SPLINE
SPL {X  -153.420, Y  +337.122, Z    +0.000, E1  +333.501, E3 -340615.542}
SPL {X  -157.288, Y  +353.220, Z    +0.000, E1  +341.134, E3 -340627.588}
SPL {X  -159.049, Y  +365.172, Z    +0.000, E1  +347.392, E3 -340633.141}
SPL {X  -159.749, Y  +373.719, Z    +0.000, E1  +352.250, E3 -340635.761}
SPL {X  -159.988, Y  +381.741, Z    +0.000, E1  +357.172, E3 -340637.236}
SPL {X  -159.990, Y  +387.352, Z    +0.000, E1  +361.387, E3 -340637.938}
SPL {X  -159.990, Y  +391.188, Z    +0.000, E1  +365.082, E3 -340638.479}
SPL {X  -159.990, Y  +395.106, Z    +0.000, E1  +369.154, E3 -340639.220}
SPL {X  -159.990, Y  +400.303, Z    +0.000, E1  +374.927, E3 -340640.541}
SPL {X  -159.990, Y  +408.423, Z    +0.000, E1  +383.302, E3 -340643.621}
SPL {X  -159.990, Y  +438.418, Z    +0.000, E1  +401.067, E3 -340665.193}
SPL {X  -159.990, Y  +482.913, Z    +0.000, E1  +407.036, E3 -340724.548}
SPL {X  -159.990, Y  +489.230, Z    +0.000, E1  +407.019, E3 -340737.059}
SPL {X  -159.990, Y  +495.241, Z    +0.000, E1  +407.026, E3 -340748.938}
SPL {X  -159.990, Y  +502.770, Z    +0.000, E1  +407.054, E3 -340763.761}
SPL {X  -159.990, Y  +511.332, Z    +0.000, E1  +407.054, E3 -340780.690}
SPL {X  -159.990, Y  +518.043, Z    +0.000, E1  +407.016, E3 -340794.030}
SPL {X  -159.990, Y  +525.485, Z    +0.000, E1  +407.063, E3 -340808.674}
SPL {X  -159.990, Y  +533.771, Z    +0.000, E1  +407.034, E3 -340825.104}
SPL {X  -159.990, Y  +542.379, Z    +0.000, E1  +407.067, E3 -340842.074}
SPL {X  -159.990, Y  +549.846, Z    +0.000, E1  +407.016, E3 -340856.919}
SPL {X  -159.990, Y  +554.843, Z    +0.000, E1  +407.014, E3 -340866.797}
SPL {X  -159.990, Y  +560.453, Z    +0.000, E1  +407.023, E3 -340877.880}
SPL {X  -159.990, Y  +566.612, Z    +0.000, E1  +407.022, E3 -340890.063}
SPL {X  -159.990, Y  +572.901, Z    +0.000, E1  +407.028, E3 -340902.474}
SPL {X  -159.990, Y  +578.640, Z    +0.000, E1  +407.021, E3 -340913.826}
SPL {X  -159.990, Y  +584.969, Z    +0.000, E1  +407.043, E3 -340926.308}
SPL {X  -159.990, Y  +591.074, Z    +0.000, E1  +407.017, E3 -340938.398}
SPL {X  -159.990, Y  +596.627, Z    +0.000, E1  +407.034, E3 -340949.343}
SPL {X  -159.990, Y  +602.039, Z    +0.000, E1  +407.021, E3 -340960.050}
SPL {X  -159.990, Y  +607.106, Z    +0.000, E1  +407.028, E3 -340970.057}
SPL {X  -159.990, Y  +612.418, Z    +0.000, E1  +407.023, E3 -340980.569}
SPL {X  -159.990, Y  +618.496, Z    +0.000, E1  +407.049, E3 -340992.535}
SPL {X  -159.990, Y  +624.357, Z    +0.000, E1  +407.020, E3 -341004.161}
SPL {X  -159.990, Y  +629.711, Z    +0.000, E1  +407.034, E3 -341014.730}
SPL {X  -159.990, Y  +635.041, Z    +0.000, E1  +407.022, E3 -341025.275}
SPL {X  -159.990, Y  +639.998, Z    +0.000, E1  +407.027, E3 -341035.067}
SPL {X  -159.990, Y  +646.188, Z    +0.000, E1  +407.041, E3 -341047.293}
SPL {X  -159.990, Y  +652.067, Z    +0.000, E1  +407.023, E3 -341058.929}
SPL {X  -159.990, Y  +657.109, Z    +0.000, E1  +407.025, E3 -341068.908}
SPL {X  -159.990, Y  +662.651, Z    +0.000, E1  +407.027, E3 -341079.864}
SPL {X  -159.990, Y  +668.015, Z    +0.000, E1  +407.025, E3 -341090.464}
SPL {X  -159.972, Y  +673.909, Z    +0.000, E1  +407.029, E3 -341102.130}
SPL {X  -159.776, Y  +679.772, Z    +0.000, E1  +406.992, E3 -341113.931}
SPL {X  -159.384, Y  +685.411, Z    +0.000, E1  +406.921, E3 -341125.492}
SPL {X  -158.642, Y  +692.228, Z    +0.000, E1  +406.819, E3 -341139.707}
SPL {X  -157.651, Y  +698.760, Z    +0.000, E1  +406.609, E3 -341153.702}
SPL {X  -156.719, Y  +703.686, Z    +0.000, E1  +406.438, E3 -341164.395}
SPL {X  -155.432, Y  +709.417, Z    +0.000, E1  +406.234, E3 -341177.039}
SPL {X  -154.084, Y  +714.570, Z    +0.000, E1  +405.932, E3 -341188.701}
SPL {X  -152.913, Y  +718.557, Z    +0.000, E1  +405.729, E3 -341197.753}
SPL {X  -151.262, Y  +723.621, Z    +0.000, E1  +405.429, E3 -341209.419}
SPL {X  -149.964, Y  +727.247, Z    +0.000, E1  +405.152, E3 -341217.924}
SPL {X  -148.611, Y  +730.759, Z    +0.000, E1  +404.909, E3 -341226.185}
SPL {X  -142.546, Y  +744.145, Z    +0.000, E1  +401.000, E3 -341286.375}
ENDSPLINE

SPLINE
SPL {X  -146.166, Y  +736.557, Z    +0.000, E1  +395.148, E3 -341330.340}
SPL {X  -153.596, Y  +716.277, Z    +0.000, E1  +386.138, E3 -341363.587}
SPL {X  -158.253, Y  +695.011, Z    +0.000, E1  +375.913, E3 -341376.697}
SPL {X  -159.486, Y  +684.192, Z    +0.000, E1  +369.965, E3 -341380.643}
SPL {X  -159.898, Y  +676.924, Z    +0.000, E1  +365.683, E3 -341382.341}
SPL {X  -159.990, Y  +671.720, Z    +0.000, E1  +362.298, E3 -341383.181}
SPL {X  -159.990, Y  +668.164, Z    +0.000, E1  +359.695, E3 -341383.597}
SPL {X  -159.990, Y  +665.062, Z    +0.000, E1  +356.961, E3 -341383.936}
SPL {X  -159.990, Y  +660.795, Z    +0.000, E1  +352.651, E3 -341384.599}
SPL {X  -159.990, Y  +654.574, Z    +0.000, E1  +345.673, E3 -341386.054}
SPL {X  -159.990, Y  +644.002, Z    +0.000, E1  +334.724, E3 -341390.251}
SPL {X  -159.990, Y  +611.706, Z    +0.000, E1  +317.244, E3 -341414.673}
SPL {X  -159.990, Y  +567.814, Z    +0.000, E1  +312.360, E3 -341474.762}
SPL {X  -159.990, Y  +558.774, Z    +0.000, E1  +312.384, E3 -341492.328}
SPL {X  -159.990, Y  +550.551, Z    +0.000, E1  +312.385, E3 -341508.269}
SPL {X  -159.990, Y  +542.502, Z    +0.000, E1  +312.392, E3 -341523.884}
SPL {X  -159.990, Y  +534.538, Z    +0.000, E1  +312.385, E3 -341539.288}
SPL {X  -159.990, Y  +527.222, Z    +0.000, E1  +312.401, E3 -341553.496}
SPL {X  -159.990, Y  +520.237, Z    +0.000, E1  +312.390, E3 -341567.027}
SPL {X  -159.990, Y  +512.328, Z    +0.000, E1  +312.388, E3 -341582.360}
SPL {X  -159.990, Y  +505.755, Z    +0.000, E1  +312.413, E3 -341595.137}
ENDSPLINE

SPLINE
SPL {X  -159.990, Y  +517.758, Z    +0.000, E1  +318.109, E3 -341602.860}
ENDSPLINE

SPLINE
SPL {X  -159.990, Y  +516.975, Z    +0.000, E1  +319.588, E3 -341613.924}
SPL {X  -159.990, Y  +508.583, Z    +0.000, E1  +318.552, E3 -341628.229}
SPL {X  -159.990, Y  +499.983, Z    +0.000, E1  +317.561, E3 -341642.683}
SPL {X  -159.990, Y  +490.062, Z    +0.000, E1  +316.490, E3 -341658.967}
SPL {X  -159.990, Y  +479.678, Z    +0.000, E1  +315.383, E3 -341675.187}
SPL {X  -159.990, Y  +468.709, Z    +0.000, E1  +314.219, E3 -341691.425}
SPL {X  -159.990, Y  +457.446, Z    +0.000, E1  +313.017, E3 -341707.078}
SPL {X  -159.990, Y  +445.780, Z    +0.000, E1  +311.870, E3 -341722.927}
ENDSPLINE

SPLINE
SPL {X  -159.990, Y  +461.496, Z    +0.000, E1  +319.836, E3 -341735.516}
ENDSPLINE

SPLINE
SPL {X  -159.990, Y  +456.934, Z    +0.000, E1  +319.854, E3 -341747.065}
SPL {X  -159.990, Y  +452.940, Z    +0.000, E1  +319.854, E3 -341757.110}
SPL {X  -159.990, Y  +448.856, Z    +0.000, E1  +319.859, E3 -341767.393}
SPL {X  -159.990, Y  +444.973, Z    +0.000, E1  +319.856, E3 -341777.159}
SPL {X  -159.990, Y  +439.927, Z    +0.000, E1  +319.837, E3 -341789.815}
SPL {X  -159.990, Y  +435.246, Z    +0.000, E1  +319.853, E3 -341801.624}
SPL {X  -159.990, Y  +430.690, Z    +0.000, E1  +319.854, E3 -341813.086}
SPL {X  -159.990, Y  +426.145, Z    +0.000, E1  +319.853, E3 -341824.526}
SPL {X  -159.990, Y  +421.880, Z    +0.000, E1  +319.860, E3 -341835.259}
SPL {X  -159.990, Y  +416.246, Z    +0.000, E1  +319.819, E3 -341849.388}
SPL {X  -159.990, Y  +409.936, Z    +0.000, E1  +319.849, E3 -341865.324}
SPL {X  -159.990, Y  +404.988, Z    +0.000, E1  +319.861, E3 -341877.790}
SPL {X  -159.990, Y  +400.535, Z    +0.000, E1  +319.859, E3 -341888.988}
SPL {X  -159.990, Y  +396.024, Z    +0.000, E1  +319.860, E3 -341900.344}
SPL {X  -159.990, Y  +391.614, Z    +0.000, E1  +319.860, E3 -341911.438}
SPL {X  -159.990, Y  +387.212, Z    +0.000, E1  +319.859, E3 -341922.510}
SPL {X  -159.990, Y  +382.743, Z    +0.000, E1  +319.857, E3 -341933.751}
SPL {X  -159.925, Y  +377.946, Z    +0.000, E1  +319.864, E3 -341945.888}
SPL {X  -159.703, Y  +372.915, Z    +0.000, E1  +319.904, E3 -341958.788}
SPL {X  -159.358, Y  +368.290, Z    +0.000, E1  +319.961, E3 -341970.751}
SPL {X  -158.955, Y  +364.333, Z    +0.000, E1  +320.046, E3 -341981.153}
SPL {X  -158.482, Y  +360.589, Z    +0.000, E1  +320.125, E3 -341991.079}
SPL {X  -157.729, Y  +355.695, Z    +0.000, E1  +320.237, E3 -342004.152}
SPL {X  -156.893, Y  +351.173, Z    +0.000, E1  +320.410, E3 -342016.435}
SPL {X  -156.148, Y  +347.650, Z    +0.000, E1  +320.549, E3 -342026.081}
SPL {X  -155.268, Y  +343.918, Z    +0.000, E1  +320.696, E3 -342036.362}
SPL {X  -153.936, Y  +338.906, Z    +0.000, E1  +320.911, E3 -342050.301}
SPL {X  -152.628, Y  +334.526, Z    +0.000, E1  +321.188, E3 -342062.703}
SPL {X  -151.010, Y  +329.654, Z    +0.000, E1  +326.674, E3 -342120.539}
ENDSPLINE

SPLINE
SPL {X  -157.513, Y  +354.453, Z    +0.000, E1  +340.941, E3 -342166.573}
SPL {X  -159.408, Y  +368.861, Z    +0.000, E1  +348.865, E3 -342175.996}
SPL {X  -159.941, Y  +378.532, Z    +0.000, E1  +354.551, E3 -342179.602}
SPL {X  -159.990, Y  +383.966, Z    +0.000, E1  +358.149, E3 -342181.054}
SPL {X  -159.990, Y  +388.001, Z    +0.000, E1  +361.086, E3 -342181.989}
SPL {X  -159.990, Y  +392.647, Z    +0.000, E1  +364.974, E3 -342183.128}
SPL {X  -159.990, Y  +397.943, Z    +0.000, E1  +369.963, E3 -342184.712}
SPL {X  -159.990, Y  +407.689, Z    +0.000, E1  +378.860, E3 -342189.367}
SPL {X  -159.990, Y  +434.822, Z    +0.000, E1  +394.625, E3 -342213.910}
SPL {X  -159.990, Y  +460.330, Z    +0.000, E1  +398.908, E3 -342258.186}
SPL {X  -159.990, Y  +464.953, Z    +0.000, E1  +398.907, E3 -342270.344}
SPL {X  -159.990, Y  +469.353, Z    +0.000, E1  +398.902, E3 -342281.925}
SPL {X  -159.990, Y  +473.222, Z    +0.000, E1  +398.891, E3 -342292.133}
SPL {X  -159.990, Y  +477.957, Z    +0.000, E1  +398.922, E3 -342304.538}
SPL {X  -159.990, Y  +482.463, Z    +0.000, E1  +398.891, E3 -342316.426}
SPL {X  -159.990, Y  +486.996, Z    +0.000, E1  +398.928, E3 -342328.258}
SPL {X  -159.990, Y  +492.629, Z    +0.000, E1  +398.922, E3 -342343.065}
SPL {X  -159.990, Y  +497.431, Z    +0.000, E1  +398.905, E3 -342355.731}
SPL {X  -159.990, Y  +502.093, Z    +0.000, E1  +398.909, E3 -342368.006}
SPL {X  -159.990, Y  +506.629, Z    +0.000, E1  +398.900, E3 -342379.938}
SPL {X  -159.990, Y  +512.483, Z    +0.000, E1  +398.947, E3 -342395.267}
SPL {X  -159.990, Y  +518.435, Z    +0.000, E1  +398.905, E3 -342410.980}
SPL {X  -159.990, Y  +523.478, Z    +0.000, E1  +398.918, E3 -342424.209}
SPL {X  -159.990, Y  +528.627, Z    +0.000, E1  +398.910, E3 -342437.762}
SPL {X  -159.990, Y  +533.053, Z    +0.000, E1  +398.899, E3 -342449.420}
SPL {X  -159.990, Y  +537.174, Z    +0.000, E1  +398.910, E3 -342460.234}
SPL {X  -159.990, Y  +541.259, Z    +0.000, E1  +398.888, E3 -342471.034}
SPL {X  -159.990, Y  +545.676, Z    +0.000, E1  +398.913, E3 -342482.605}
SPL {X  -159.990, Y  +550.777, Z    +0.000, E1  +398.906, E3 -342496.024}
SPL {X  -159.990, Y  +556.271, Z    +0.000, E1  +398.927, E3 -342510.426}
SPL {X  -159.990, Y  +561.696, Z    +0.000, E1  +398.912, E3 -342524.696}
SPL {X  -159.990, Y  +566.650, Z    +0.000, E1  +398.917, E3 -342537.710}
SPL {X  -159.990, Y  +571.814, Z    +0.000, E1  +398.914, E3 -342551.312}
SPL {X  -159.990, Y  +576.364, Z    +0.000, E1  +398.896, E3 -342563.316}
SPL {X  -159.990, Y  +582.060, Z    +0.000, E1  +398.942, E3 -342578.221}
SPL {X  -159.990, Y  +587.761, Z    +0.000, E1  +398.902, E3 -342593.270}
SPL {X  -159.990, Y  +592.962, Z    +0.000, E1  +398.925, E3 -342606.914}
SPL {X  -159.990, Y  +597.767, Z    +0.000, E1  +398.897, E3 -342619.589}
SPL {X  -159.990, Y  +602.727, Z    +0.000, E1  +398.920, E3 -342632.600}
SPL {X  -159.990, Y  +608.112, Z    +0.000, E1  +398.911, E3 -342646.775}
SPL {X  -159.990, Y  +613.039, Z    +0.000, E1  +398.906, E3 -342659.737}
SPL {X  -159.990, Y  +618.087, Z    +0.000, E1  +398.915, E3 -342672.996}
SPL {X  -159.990, Y  +623.264, Z    +0.000, E1  +398.906, E3 -342686.631}
SPL {X  -159.990, Y  +628.669, Z    +0.000, E1  +398.928, E3 -342700.799}
SPL {X  -159.990, Y  +634.089, Z    +0.000, E1  +398.907, E3 -342715.075}
SPL {X  -159.990, Y  +638.639, Z    +0.000, E1  +398.904, E3 -342727.060}
SPL {X  -159.990, Y  +644.750, Z    +0.000, E1  +398.946, E3 -342743.065}
SPL {X  -159.990, Y  +650.458, Z    +0.000, E1  +398.900, E3 -342758.138}
SPL {X  -159.990, Y  +654.813, Z    +0.000, E1  +398.905, E3 -342769.582}
SPL {X  -159.990, Y  +660.353, Z    +0.000, E1  +398.930, E3 -342784.113}
SPL {X  -159.990, Y  +665.703, Z    +0.000, E1  +398.903, E3 -342798.221}
SPL {X  -159.990, Y  +669.966, Z    +0.000, E1  +398.902, E3 -342809.427}
SPL {X  -159.954, Y  +674.895, Z    +0.000, E1  +398.910, E3 -342822.407}
SPL {X  -159.761, Y  +680.061, Z    +0.000, E1  +398.873, E3 -342836.186}
SPL {X  -159.443, Y  +684.716, Z    +0.000, E1  +398.815, E3 -342848.751}
SPL {X  -158.962, Y  +689.604, Z    +0.000, E1  +398.740, E3 -342862.121}
SPL {X  -158.318, Y  +694.567, Z    +0.000, E1  +398.614, E3 -342875.882}
SPL {X  -157.472, Y  +699.775, Z    +0.000, E1  +398.483, E3 -342890.441}
SPL {X  -156.506, Y  +704.705, Z    +0.000, E1  +398.294, E3 -342904.442}
SPL {X  -155.680, Y  +708.387, Z    +0.000, E1  +398.127, E3 -342915.013}
SPL {X  -154.586, Y  +712.730, Z    +0.000, E1  +397.967, E3 -342927.510}
SPL {X  -153.345, Y  +717.131, Z    +0.000, E1  +397.713, E3 -342940.394}
SPL {X  -151.080, Y  +724.146, Z    +0.000, E1  +393.201, E3 -342998.847}
ENDSPLINE

SPLINE
SPL {X  -157.921, Y  +697.149, Z    +0.000, E1  +377.701, E3 -343050.408}
SPL {X  -159.579, Y  +682.959, Z    +0.000, E1  +369.793, E3 -343058.357}
SPL {X  -159.938, Y  +675.561, Z    +0.000, E1  +365.399, E3 -343060.779}
SPL {X  -159.990, Y  +669.910, Z    +0.000, E1  +361.710, E3 -343062.070}
SPL {X  -159.990, Y  +665.465, Z    +0.000, E1  +358.378, E3 -343062.987}
SPL {X  -159.990, Y  +661.791, Z    +0.000, E1  +355.213, E3 -343063.825}
SPL {X  -159.990, Y  +656.991, Z    +0.000, E1  +350.742, E3 -343065.244}
SPL {X  -159.990, Y  +648.067, Z    +0.000, E1  +342.328, E3 -343068.974}
SPL {X  -159.990, Y  +620.451, Z    +0.000, E1  +325.419, E3 -343092.821}
SPL {X  -159.990, Y  +591.256, Z    +0.000, E1  +319.966, E3 -343139.314}
SPL {X  -159.990, Y  +586.740, Z    +0.000, E1  +319.956, E3 -343150.705}
SPL {X  -159.990, Y  +581.814, Z    +0.000, E1  +319.956, E3 -343163.144}
SPL {X  -159.990, Y  +577.274, Z    +0.000, E1  +319.964, E3 -343174.622}
SPL {X  -159.990, Y  +572.933, Z    +0.000, E1  +319.959, E3 -343185.563}
SPL {X  -159.990, Y  +568.504, Z    +0.000, E1  +319.956, E3 -343196.725}
SPL {X  -159.990, Y  +563.189, Z    +0.000, E1  +319.932, E3 -343210.099}
SPL {X  -159.990, Y  +557.707, Z    +0.000, E1  +319.949, E3 -343223.954}
SPL {X  -159.990, Y  +553.571, Z    +0.000, E1  +319.954, E3 -343234.373}
SPL {X  -159.990, Y  +549.413, Z    +0.000, E1  +319.938, E3 -343244.839}
SPL {X  -159.990, Y  +543.439, Z    +0.000, E1  +319.921, E3 -343259.926}
SPL {X  -159.990, Y  +537.213, Z    +0.000, E1  +319.937, E3 -343275.669}
SPL {X  -159.990, Y  +532.291, Z    +0.000, E1  +319.951, E3 -343288.094}
SPL {X  -159.990, Y  +528.899, Z    +0.000, E1  +319.955, E3 -343296.647}
SPL {X  -159.990, Y  +523.984, Z    +0.000, E1  +319.922, E3 -343308.993}
SPL {X  -159.990, Y  +496.806, Z    +0.000, E1  +312.216, E3 -343322.908}
SPL {X  -159.990, Y  +490.245, Z    +0.000, E1  +312.831, E3 -343339.439}
SPL {X  -159.990, Y  +484.831, Z    +0.000, E1  +314.066, E3 -343357.672}
SPL {X  -159.990, Y  +480.580, Z    +0.000, E1  +315.242, E3 -343373.358}
SPL {X  -159.990, Y  +476.546, Z    +0.000, E1  +316.165, E3 -343387.653}
SPL {X  -159.990, Y  +473.377, Z    +0.000, E1  +316.953, E3 -343399.268}
SPL {X  -159.990, Y  +470.788, Z    +0.000, E1  +317.853, E3 -343410.681}
SPL {X  -159.990, Y  +467.944, Z    +0.000, E1  +318.635, E3 -343422.002}
SPL {X  -159.990, Y  +465.057, Z    +0.000, E1  +319.375, E3 -343433.568}
SPL {X  -159.990, Y  +461.409, Z    +0.000, E1  +319.848, E3 -343445.467}
SPL {X  -159.990, Y  +456.934, Z    +0.000, E1  +319.854, E3 -343456.743}
SPL {X  -159.990, Y  +452.940, Z    +0.000, E1  +319.854, E3 -343466.787}
SPL {X  -159.990, Y  +448.856, Z    +0.000, E1  +319.859, E3 -343477.071}
SPL {X  -159.990, Y  +444.973, Z    +0.000, E1  +319.856, E3 -343486.836}
SPL {X  -159.990, Y  +439.927, Z    +0.000, E1  +319.837, E3 -343499.492}
SPL {X  -159.990, Y  +435.246, Z    +0.000, E1  +319.853, E3 -343511.302}
SPL {X  -159.990, Y  +430.690, Z    +0.000, E1  +319.854, E3 -343522.763}
SPL {X  -159.990, Y  +426.145, Z    +0.000, E1  +319.853, E3 -343534.203}
SPL {X  -159.990, Y  +421.880, Z    +0.000, E1  +319.860, E3 -343544.936}
SPL {X  -159.990, Y  +416.246, Z    +0.000, E1  +319.819, E3 -343559.065}
SPL {X  -159.990, Y  +409.936, Z    +0.000, E1  +319.849, E3 -343575.002}
SPL {X  -159.990, Y  +404.988, Z    +0.000, E1  +319.861, E3 -343587.467}
SPL {X  -159.990, Y  +400.535, Z    +0.000, E1  +319.859, E3 -343598.665}
SPL {X  -159.990, Y  +396.024, Z    +0.000, E1  +319.860, E3 -343610.021}
SPL {X  -159.990, Y  +391.614, Z    +0.000, E1  +319.860, E3 -343621.115}
SPL {X  -159.990, Y  +387.212, Z    +0.000, E1  +319.859, E3 -343632.187}
SPL {X  -159.990, Y  +382.743, Z    +0.000, E1  +319.857, E3 -343643.429}
SPL {X  -159.925, Y  +377.946, Z    +0.000, E1  +319.864, E3 -343655.566}
SPL {X  -159.703, Y  +372.915, Z    +0.000, E1  +319.904, E3 -343668.465}
SPL {X  -159.358, Y  +368.290, Z    +0.000, E1  +319.961, E3 -343680.428}
SPL {X  -158.955, Y  +364.333, Z    +0.000, E1  +320.046, E3 -343690.830}
SPL {X  -158.482, Y  +360.589, Z    +0.000, E1  +320.125, E3 -343700.757}
SPL {X  -157.729, Y  +355.695, Z    +0.000, E1  +320.237, E3 -343713.829}
SPL {X  -156.893, Y  +351.173, Z    +0.000, E1  +320.410, E3 -343726.113}
SPL {X  -156.148, Y  +347.650, Z    +0.000, E1  +320.549, E3 -343735.759}
SPL {X  -155.268, Y  +343.918, Z    +0.000, E1  +320.696, E3 -343746.039}
SPL {X  -154.153, Y  +339.677, Z    +0.000, E1  +320.896, E3 -343757.846}
SPL {X  -152.885, Y  +335.352, Z    +0.000, E1  +321.114, E3 -343770.000}
SPL {X  -151.010, Y  +329.654, Z    +0.000, E1  +326.674, E3 -343830.217}
ENDSPLINE

SPLINE
SPL {X  -157.513, Y  +354.453, Z    +0.000, E1  +340.941, E3 -343876.251}
SPL {X  -159.408, Y  +368.861, Z    +0.000, E1  +348.865, E3 -343885.674}
SPL {X  -159.941, Y  +378.532, Z    +0.000, E1  +354.551, E3 -343889.279}
SPL {X  -159.990, Y  +383.966, Z    +0.000, E1  +358.149, E3 -343890.731}
SPL {X  -159.990, Y  +389.165, Z    +0.000, E1  +361.929, E3 -343891.933}
SPL {X  -159.990, Y  +396.368, Z    +0.000, E1  +368.359, E3 -343893.905}
SPL {X  -159.990, Y  +407.689, Z    +0.000, E1  +378.860, E3 -343899.044}
SPL {X  -159.990, Y  +434.822, Z    +0.000, E1  +394.625, E3 -343923.588}
SPL {X  -159.990, Y  +460.330, Z    +0.000, E1  +398.908, E3 -343967.863}
SPL {X  -159.990, Y  +464.953, Z    +0.000, E1  +398.907, E3 -343980.022}
SPL {X  -159.990, Y  +469.353, Z    +0.000, E1  +398.902, E3 -343991.602}
SPL {X  -159.990, Y  +473.222, Z    +0.000, E1  +398.891, E3 -344001.811}
SPL {X  -159.990, Y  +477.957, Z    +0.000, E1  +398.922, E3 -344014.216}
SPL {X  -159.990, Y  +482.463, Z    +0.000, E1  +398.891, E3 -344026.103}
SPL {X  -159.990, Y  +486.996, Z    +0.000, E1  +398.928, E3 -344037.935}
SPL {X  -159.990, Y  +492.629, Z    +0.000, E1  +398.922, E3 -344052.742}
SPL {X  -159.990, Y  +497.431, Z    +0.000, E1  +398.905, E3 -344065.408}
SPL {X  -159.990, Y  +502.093, Z    +0.000, E1  +398.909, E3 -344077.683}
SPL {X  -159.990, Y  +507.821, Z    +0.000, E1  +398.930, E3 -344092.703}
SPL {X  -159.990, Y  +513.533, Z    +0.000, E1  +398.910, E3 -344107.762}
SPL {X  -159.990, Y  +518.435, Z    +0.000, E1  +398.905, E3 -344120.658}
SPL {X  -159.990, Y  +523.478, Z    +0.000, E1  +398.918, E3 -344133.886}
SPL {X  -159.990, Y  +528.627, Z    +0.000, E1  +398.910, E3 -344147.440}
SPL {X  -159.990, Y  +533.053, Z    +0.000, E1  +398.899, E3 -344159.097}
SPL {X  -159.990, Y  +537.174, Z    +0.000, E1  +398.910, E3 -344169.912}
SPL {X  -159.990, Y  +542.636, Z    +0.000, E1  +398.920, E3 -344184.280}
SPL {X  -159.990, Y  +549.483, Z    +0.000, E1  +398.950, E3 -344202.235}
SPL {X  -159.990, Y  +556.271, Z    +0.000, E1  +398.927, E3 -344220.104}
SPL {X  -159.990, Y  +561.696, Z    +0.000, E1  +398.912, E3 -344234.373}
SPL {X  -159.990, Y  +566.650, Z    +0.000, E1  +398.917, E3 -344247.387}
SPL {X  -159.990, Y  +571.814, Z    +0.000, E1  +398.914, E3 -344260.990}
SPL {X  -159.990, Y  +576.364, Z    +0.000, E1  +398.896, E3 -344272.993}
SPL {X  -159.990, Y  +582.060, Z    +0.000, E1  +398.942, E3 -344287.898}
SPL {X  -159.990, Y  +589.106, Z    +0.000, E1  +398.939, E3 -344306.430}
SPL {X  -159.990, Y  +596.185, Z    +0.000, E1  +398.945, E3 -344325.039}
SPL {X  -159.990, Y  +602.727, Z    +0.000, E1  +398.920, E3 -344342.278}
SPL {X  -159.990, Y  +608.112, Z    +0.000, E1  +398.911, E3 -344356.452}
SPL {X  -159.990, Y  +613.039, Z    +0.000, E1  +398.906, E3 -344369.415}
SPL {X  -159.990, Y  +618.087, Z    +0.000, E1  +398.915, E3 -344382.673}
SPL {X  -159.990, Y  +623.264, Z    +0.000, E1  +398.906, E3 -344396.308}
SPL {X  -159.990, Y  +627.067, Z    +0.000, E1  +398.891, E3 -344406.328}
SPL {X  -159.990, Y  +630.187, Z    +0.000, E1  +398.892, E3 -344414.515}
SPL {X  -159.990, Y  +634.089, Z    +0.000, E1  +398.907, E3 -344424.752}
SPL {X  -159.990, Y  +638.639, Z    +0.000, E1  +398.904, E3 -344436.738}
SPL {X  -159.990, Y  +643.555, Z    +0.000, E1  +398.910, E3 -344449.657}
SPL {X  -159.990, Y  +649.380, Z    +0.000, E1  +398.930, E3 -344464.935}
SPL {X  -159.990, Y  +654.813, Z    +0.000, E1  +398.905, E3 -344479.260}
SPL {X  -159.990, Y  +658.715, Z    +0.000, E1  +398.892, E3 -344489.541}
SPL {X  -159.990, Y  +661.848, Z    +0.000, E1  +398.892, E3 -344497.779}
SPL {X  -159.990, Y  +665.703, Z    +0.000, E1  +398.903, E3 -344507.898}
SPL {X  -159.990, Y  +669.966, Z    +0.000, E1  +398.902, E3 -344519.105}
SPL {X  -159.954, Y  +674.895, Z    +0.000, E1  +398.910, E3 -344532.085}
SPL {X  -159.761, Y  +680.061, Z    +0.000, E1  +398.873, E3 -344545.864}
SPL {X  -159.443, Y  +684.716, Z    +0.000, E1  +398.815, E3 -344558.429}
SPL {X  -158.962, Y  +689.604, Z    +0.000, E1  +398.740, E3 -344571.798}
SPL {X  -158.139, Y  +695.766, Z    +0.000, E1  +398.623, E3 -344588.844}
SPL {X  -157.275, Y  +700.848, Z    +0.000, E1  +398.415, E3 -344603.196}
SPL {X  -156.506, Y  +704.705, Z    +0.000, E1  +398.294, E3 -344614.119}
SPL {X  -155.357, Y  +709.721, Z    +0.000, E1  +398.108, E3 -344628.474}
SPL {X  -154.286, Y  +713.838, Z    +0.000, E1  +397.877, E3 -344640.457}
SPL {X  -153.345, Y  +717.131, Z    +0.000, E1  +397.713, E3 -344650.071}
SPL {X  -151.080, Y  +724.146, Z    +0.000, E1  +393.201, E3 -344708.525}
ENDSPLINE

SPLINE
SPL {X  -157.921, Y  +697.149, Z    +0.000, E1  +377.701, E3 -344760.086}
SPL {X  -159.579, Y  +682.959, Z    +0.000, E1  +369.793, E3 -344768.034}
SPL {X  -159.938, Y  +675.561, Z    +0.000, E1  +365.399, E3 -344770.456}
SPL {X  -159.990, Y  +669.910, Z    +0.000, E1  +361.710, E3 -344771.747}
SPL {X  -159.990, Y  +665.465, Z    +0.000, E1  +358.378, E3 -344772.664}
SPL {X  -159.990, Y  +661.791, Z    +0.000, E1  +355.213, E3 -344773.502}
SPL {X  -159.990, Y  +656.991, Z    +0.000, E1  +350.742, E3 -344774.921}
SPL {X  -159.990, Y  +648.067, Z    +0.000, E1  +342.328, E3 -344778.651}
SPL {X  -159.990, Y  +624.891, Z    +0.000, E1  +327.004, E3 -344797.139}
SPL {X  -159.990, Y  +618.109, Z    +0.000, E1  +324.631, E3 -344805.315}
SPL {X  -159.990, Y  +591.256, Z    +0.000, E1  +319.966, E3 -344848.992}
SPL {X  -159.990, Y  +586.740, Z    +0.000, E1  +319.956, E3 -344860.382}
SPL {X  -159.990, Y  +581.814, Z    +0.000, E1  +319.956, E3 -344872.821}
SPL {X  -159.990, Y  +577.274, Z    +0.000, E1  +319.964, E3 -344884.299}
SPL {X  -159.990, Y  +572.933, Z    +0.000, E1  +319.959, E3 -344895.240}
SPL {X  -159.990, Y  +568.504, Z    +0.000, E1  +319.956, E3 -344906.403}
SPL {X  -159.990, Y  +564.427, Z    +0.000, E1  +319.959, E3 -344916.689}
SPL {X  -159.990, Y  +558.823, Z    +0.000, E1  +319.916, E3 -344930.768}
SPL {X  -159.990, Y  +553.571, Z    +0.000, E1  +319.954, E3 -344944.050}
SPL {X  -159.990, Y  +549.413, Z    +0.000, E1  +319.938, E3 -344954.516}
SPL {X  -159.990, Y  +543.439, Z    +0.000, E1  +319.921, E3 -344969.604}
SPL {X  -159.990, Y  +537.213, Z    +0.000, E1  +319.937, E3 -344985.347}
SPL {X  -159.990, Y  +532.291, Z    +0.000, E1  +319.951, E3 -344997.772}
SPL {X  -159.990, Y  +527.393, Z    +0.000, E1  +319.924, E3 -345010.081}
SPL {X  -159.990, Y  +522.533, Z    +0.000, E1  +319.951, E3 -345022.378}
SPL {X  -159.990, Y  +502.378, Z    +0.000, E1  +313.079, E3 -345026.782}
SPL {X  -159.990, Y  +493.568, Z    +0.000, E1  +312.053, E3 -345037.950}
SPL {X  -159.990, Y  +489.464, Z    +0.000, E1  +313.059, E3 -345051.816}
SPL {X  -159.990, Y  +484.831, Z    +0.000, E1  +314.066, E3 -345067.350}
SPL {X  -159.990, Y  +480.580, Z    +0.000, E1  +315.242, E3 -345083.036}
SPL {X  -159.990, Y  +476.546, Z    +0.000, E1  +316.165, E3 -345097.331}
SPL {X  -159.990, Y  +472.671, Z    +0.000, E1  +317.192, E3 -345112.158}
SPL {X  -159.990, Y  +468.809, Z    +0.000, E1  +318.343, E3 -345128.087}
SPL {X  -159.990, Y  +465.057, Z    +0.000, E1  +319.375, E3 -345143.245}
SPL {X  -159.990, Y  +461.409, Z    +0.000, E1  +319.848, E3 -345155.144}
SPL {X  -159.990, Y  +456.934, Z    +0.000, E1  +319.854, E3 -345166.420}
SPL {X  -159.990, Y  +452.940, Z    +0.000, E1  +319.854, E3 -345176.465}
SPL {X  -159.990, Y  +448.856, Z    +0.000, E1  +319.859, E3 -345186.748}
SPL {X  -159.990, Y  +444.973, Z    +0.000, E1  +319.856, E3 -345196.513}
SPL {X  -159.990, Y  +439.927, Z    +0.000, E1  +319.837, E3 -345209.170}
SPL {X  -159.990, Y  +435.246, Z    +0.000, E1  +319.853, E3 -345220.979}
SPL {X  -159.990, Y  +430.690, Z    +0.000, E1  +319.854, E3 -345232.441}
SPL {X  -159.990, Y  +426.145, Z    +0.000, E1  +319.853, E3 -345243.881}
SPL {X  -159.990, Y  +421.880, Z    +0.000, E1  +319.860, E3 -345254.614}
SPL {X  -159.990, Y  +416.246, Z    +0.000, E1  +319.819, E3 -345268.742}
SPL {X  -159.990, Y  +409.936, Z    +0.000, E1  +319.849, E3 -345284.679}
SPL {X  -159.990, Y  +404.988, Z    +0.000, E1  +319.861, E3 -345297.145}
SPL {X  -159.990, Y  +400.535, Z    +0.000, E1  +319.859, E3 -345308.343}
SPL {X  -159.990, Y  +396.024, Z    +0.000, E1  +319.860, E3 -345319.699}
SPL {X  -159.990, Y  +391.614, Z    +0.000, E1  +319.860, E3 -345330.792}
SPL {X  -159.990, Y  +387.212, Z    +0.000, E1  +319.859, E3 -345341.865}
SPL {X  -159.990, Y  +382.743, Z    +0.000, E1  +319.857, E3 -345353.106}
SPL {X  -159.925, Y  +377.946, Z    +0.000, E1  +319.864, E3 -345365.243}
SPL {X  -159.703, Y  +372.915, Z    +0.000, E1  +319.904, E3 -345378.143}
SPL {X  -159.358, Y  +368.290, Z    +0.000, E1  +319.961, E3 -345390.105}
SPL {X  -158.955, Y  +364.333, Z    +0.000, E1  +320.046, E3 -345400.508}
SPL {X  -158.270, Y  +359.106, Z    +0.000, E1  +320.118, E3 -345414.319}
SPL {X  -157.143, Y  +352.453, Z    +0.000, E1  +320.322, E3 -345432.250}
SPL {X  -156.148, Y  +347.650, Z    +0.000, E1  +320.549, E3 -345445.436}
SPL {X  -155.268, Y  +343.918, Z    +0.000, E1  +320.696, E3 -345455.717}
SPL {X  -154.153, Y  +339.677, Z    +0.000, E1  +320.896, E3 -345467.524}
SPL {X  -152.885, Y  +335.352, Z    +0.000, E1  +321.114, E3 -345479.678}
SPL {X  -151.010, Y  +329.654, Z    +0.000, E1  +326.674, E3 -345539.894}
ENDSPLINE

SPLINE
SPL {X  -157.513, Y  +354.453, Z    +0.000, E1  +340.941, E3 -345585.928}
SPL {X  -159.408, Y  +368.861, Z    +0.000, E1  +348.865, E3 -345595.351}
SPL {X  -159.941, Y  +378.532, Z    +0.000, E1  +354.551, E3 -345598.957}
SPL {X  -159.990, Y  +383.966, Z    +0.000, E1  +358.149, E3 -345600.409}
SPL {X  -159.990, Y  +389.165, Z    +0.000, E1  +361.929, E3 -345601.610}
SPL {X  -159.990, Y  +394.164, Z    +0.000, E1  +366.430, E3 -345602.903}
SPL {X  -159.990, Y  +399.434, Z    +0.000, E1  +371.306, E3 -345604.663}
SPL {X  -159.990, Y  +407.956, Z    +0.000, E1  +379.215, E3 -345608.751}
SPL {X  -159.990, Y  +429.014, Z    +0.000, E1  +392.438, E3 -345626.621}
SPL {X  -159.990, Y  +437.635, Z    +0.000, E1  +395.495, E3 -345636.853}
SPL {X  -159.990, Y  +460.330, Z    +0.000, E1  +398.908, E3 -345677.541}
SPL {X  -159.990, Y  +464.953, Z    +0.000, E1  +398.907, E3 -345689.699}
SPL {X  -159.990, Y  +469.353, Z    +0.000, E1  +398.902, E3 -345701.279}
SPL {X  -159.990, Y  +473.222, Z    +0.000, E1  +398.891, E3 -345711.488}
SPL {X  -159.990, Y  +476.615, Z    +0.000, E1  +398.890, E3 -345720.423}
SPL {X  -159.990, Y  +481.308, Z    +0.000, E1  +398.917, E3 -345732.705}
SPL {X  -159.990, Y  +486.996, Z    +0.000, E1  +398.928, E3 -345747.613}
SPL {X  -159.990, Y  +492.629, Z    +0.000, E1  +398.922, E3 -345762.420}
SPL {X  -159.990, Y  +497.431, Z    +0.000, E1  +398.905, E3 -345775.086}
SPL {X  -159.990, Y  +502.093, Z    +0.000, E1  +398.909, E3 -345787.360}
SPL {X  -159.990, Y  +507.821, Z    +0.000, E1  +398.930, E3 -345802.381}
SPL {X  -159.990, Y  +513.533, Z    +0.000, E1  +398.910, E3 -345817.440}
SPL {X  -159.990, Y  +518.435, Z    +0.000, E1  +398.905, E3 -345830.335}
SPL {X  -159.990, Y  +523.478, Z    +0.000, E1  +398.918, E3 -345843.564}
SPL {X  -159.990, Y  +528.627, Z    +0.000, E1  +398.910, E3 -345857.117}
SPL {X  -159.990, Y  +534.392, Z    +0.000, E1  +398.932, E3 -345872.247}
SPL {X  -159.990, Y  +540.299, Z    +0.000, E1  +398.912, E3 -345887.822}
SPL {X  -159.990, Y  +545.676, Z    +0.000, E1  +398.913, E3 -345901.960}
SPL {X  -159.990, Y  +550.777, Z    +0.000, E1  +398.906, E3 -345915.379}
SPL {X  -159.990, Y  +556.271, Z    +0.000, E1  +398.927, E3 -345929.781}
SPL {X  -159.990, Y  +561.696, Z    +0.000, E1  +398.912, E3 -345944.051}
SPL {X  -159.990, Y  +566.650, Z    +0.000, E1  +398.917, E3 -345957.064}
SPL {X  -159.990, Y  +571.814, Z    +0.000, E1  +398.914, E3 -345970.667}
SPL {X  -159.990, Y  +576.364, Z    +0.000, E1  +398.896, E3 -345982.670}
SPL {X  -159.990, Y  +582.060, Z    +0.000, E1  +398.942, E3 -345997.576}
SPL {X  -159.990, Y  +587.761, Z    +0.000, E1  +398.902, E3 -346012.625}
SPL {X  -159.990, Y  +592.962, Z    +0.000, E1  +398.925, E3 -346026.269}
SPL {X  -159.990, Y  +597.767, Z    +0.000, E1  +398.897, E3 -346038.944}
SPL {X  -159.990, Y  +602.727, Z    +0.000, E1  +398.920, E3 -346051.955}
SPL {X  -159.990, Y  +608.112, Z    +0.000, E1  +398.911, E3 -346066.130}
SPL {X  -159.990, Y  +614.125, Z    +0.000, E1  +398.936, E3 -346081.905}
SPL {X  -159.990, Y  +619.061, Z    +0.000, E1  +398.894, E3 -346094.936}
SPL {X  -159.990, Y  +623.264, Z    +0.000, E1  +398.906, E3 -346105.985}
SPL {X  -159.990, Y  +627.067, Z    +0.000, E1  +398.891, E3 -346116.005}
SPL {X  -159.990, Y  +630.187, Z    +0.000, E1  +398.892, E3 -346124.193}
SPL {X  -159.990, Y  +634.089, Z    +0.000, E1  +398.907, E3 -346134.429}
SPL {X  -159.990, Y  +638.639, Z    +0.000, E1  +398.904, E3 -346146.415}
SPL {X  -159.990, Y  +643.555, Z    +0.000, E1  +398.910, E3 -346159.335}
SPL {X  -159.990, Y  +649.380, Z    +0.000, E1  +398.930, E3 -346174.612}
SPL {X  -159.990, Y  +654.813, Z    +0.000, E1  +398.905, E3 -346188.937}
SPL {X  -159.990, Y  +658.715, Z    +0.000, E1  +398.892, E3 -346199.218}
SPL {X  -159.990, Y  +661.848, Z    +0.000, E1  +398.892, E3 -346207.456}
SPL {X  -159.990, Y  +665.703, Z    +0.000, E1  +398.903, E3 -346217.576}
SPL {X  -159.990, Y  +669.966, Z    +0.000, E1  +398.902, E3 -346228.782}
SPL {X  -159.954, Y  +674.895, Z    +0.000, E1  +398.910, E3 -346241.762}
SPL {X  -159.761, Y  +680.061, Z    +0.000, E1  +398.873, E3 -346255.541}
SPL {X  -159.443, Y  +684.716, Z    +0.000, E1  +398.815, E3 -346268.106}
SPL {X  -158.962, Y  +689.604, Z    +0.000, E1  +398.740, E3 -346281.475}
SPL {X  -158.139, Y  +695.766, Z    +0.000, E1  +398.623, E3 -346298.521}
SPL {X  -157.275, Y  +700.848, Z    +0.000, E1  +398.415, E3 -346312.873}
SPL {X  -156.506, Y  +704.705, Z    +0.000, E1  +398.294, E3 -346323.797}
SPL {X  -155.357, Y  +709.721, Z    +0.000, E1  +398.108, E3 -346338.152}
SPL {X  -154.286, Y  +713.838, Z    +0.000, E1  +397.877, E3 -346350.134}
SPL {X  -153.345, Y  +717.131, Z    +0.000, E1  +397.713, E3 -346359.748}
SPL {X  -151.080, Y  +724.146, Z    +0.000, E1  +393.201, E3 -346418.202}
ENDSPLINE

SPLINE
SPL {X  -157.921, Y  +697.149, Z    +0.000, E1  +377.701, E3 -346469.763}
SPL {X  -159.579, Y  +682.959, Z    +0.000, E1  +369.793, E3 -346477.711}
SPL {X  -159.938, Y  +675.561, Z    +0.000, E1  +365.399, E3 -346480.134}
SPL {X  -159.990, Y  +669.910, Z    +0.000, E1  +361.710, E3 -346481.424}
SPL {X  -159.990, Y  +665.465, Z    +0.000, E1  +358.378, E3 -346482.342}
SPL {X  -159.990, Y  +661.791, Z    +0.000, E1  +355.213, E3 -346483.180}
SPL {X  -159.990, Y  +656.991, Z    +0.000, E1  +350.742, E3 -346484.599}
SPL {X  -159.990, Y  +648.067, Z    +0.000, E1  +342.328, E3 -346488.328}
SPL {X  -159.990, Y  +624.891, Z    +0.000, E1  +327.004, E3 -346506.816}
SPL {X  -159.990, Y  +618.109, Z    +0.000, E1  +324.631, E3 -346514.992}
SPL {X  -159.990, Y  +591.256, Z    +0.000, E1  +319.966, E3 -346558.669}
SPL {X  -159.990, Y  +586.740, Z    +0.000, E1  +319.956, E3 -346570.059}
SPL {X  -159.990, Y  +581.814, Z    +0.000, E1  +319.956, E3 -346582.499}
SPL {X  -159.990, Y  +577.274, Z    +0.000, E1  +319.964, E3 -346593.976}
SPL {X  -159.990, Y  +572.933, Z    +0.000, E1  +319.959, E3 -346604.918}
SPL {X  -159.990, Y  +568.504, Z    +0.000, E1  +319.956, E3 -346616.080}
SPL {X  -159.990, Y  +564.427, Z    +0.000, E1  +319.959, E3 -346626.366}
SPL {X  -159.990, Y  +558.823, Z    +0.000, E1  +319.916, E3 -346640.446}
SPL {X  -159.990, Y  +553.571, Z    +0.000, E1  +319.954, E3 -346653.727}
SPL {X  -159.990, Y  +549.413, Z    +0.000, E1  +319.938, E3 -346664.193}
SPL {X  -159.990, Y  +543.439, Z    +0.000, E1  +319.921, E3 -346679.281}
SPL {X  -159.990, Y  +537.213, Z    +0.000, E1  +319.937, E3 -346695.024}
SPL {X  -159.990, Y  +532.291, Z    +0.000, E1  +319.951, E3 -346707.449}
SPL {X  -159.990, Y  +527.393, Z    +0.000, E1  +319.924, E3 -346719.758}
SPL {X  -159.990, Y  +522.533, Z    +0.000, E1  +319.951, E3 -346732.055}
SPL {X  -159.990, Y  +502.378, Z    +0.000, E1  +313.079, E3 -346736.459}
SPL {X  -159.990, Y  +493.568, Z    +0.000, E1  +312.053, E3 -346747.627}
SPL {X  -159.990, Y  +489.464, Z    +0.000, E1  +313.059, E3 -346761.494}
SPL {X  -159.990, Y  +484.831, Z    +0.000, E1  +314.066, E3 -346777.027}
SPL {X  -159.990, Y  +480.580, Z    +0.000, E1  +315.242, E3 -346792.713}
SPL {X  -159.990, Y  +476.546, Z    +0.000, E1  +316.165, E3 -346807.008}
SPL {X  -159.990, Y  +472.671, Z    +0.000, E1  +317.192, E3 -346821.835}
SPL {X  -159.990, Y  +468.809, Z    +0.000, E1  +318.343, E3 -346837.764}
SPL {X  -159.990, Y  +465.057, Z    +0.000, E1  +319.375, E3 -346852.922}
SPL {X  -159.990, Y  +461.409, Z    +0.000, E1  +319.848, E3 -346864.822}
SPL {X  -159.990, Y  +456.934, Z    +0.000, E1  +319.854, E3 -346876.097}
SPL {X  -159.990, Y  +452.940, Z    +0.000, E1  +319.854, E3 -346886.142}
SPL {X  -159.990, Y  +448.856, Z    +0.000, E1  +319.859, E3 -346896.425}
SPL {X  -159.990, Y  +444.973, Z    +0.000, E1  +319.856, E3 -346906.191}
SPL {X  -159.990, Y  +439.927, Z    +0.000, E1  +319.837, E3 -346918.847}
SPL {X  -159.990, Y  +435.246, Z    +0.000, E1  +319.853, E3 -346930.656}
SPL {X  -159.990, Y  +430.690, Z    +0.000, E1  +319.854, E3 -346942.118}
SPL {X  -159.990, Y  +426.145, Z    +0.000, E1  +319.853, E3 -346953.558}
SPL {X  -159.990, Y  +421.880, Z    +0.000, E1  +319.860, E3 -346964.291}
SPL {X  -159.990, Y  +416.246, Z    +0.000, E1  +319.819, E3 -346978.420}
SPL {X  -159.990, Y  +409.936, Z    +0.000, E1  +319.849, E3 -346994.356}
SPL {X  -159.990, Y  +404.988, Z    +0.000, E1  +319.861, E3 -347006.822}
SPL {X  -159.990, Y  +400.535, Z    +0.000, E1  +319.859, E3 -347018.020}
SPL {X  -159.990, Y  +396.024, Z    +0.000, E1  +319.860, E3 -347029.376}
SPL {X  -159.990, Y  +391.614, Z    +0.000, E1  +319.860, E3 -347040.470}
SPL {X  -159.990, Y  +387.212, Z    +0.000, E1  +319.859, E3 -347051.542}
SPL {X  -159.990, Y  +382.743, Z    +0.000, E1  +319.857, E3 -347062.784}
SPL {X  -159.925, Y  +377.946, Z    +0.000, E1  +319.864, E3 -347074.920}
SPL {X  -159.703, Y  +372.915, Z    +0.000, E1  +319.904, E3 -347087.820}
SPL {X  -159.358, Y  +368.290, Z    +0.000, E1  +319.961, E3 -347099.783}
SPL {X  -158.955, Y  +364.333, Z    +0.000, E1  +320.046, E3 -347110.185}
SPL {X  -158.270, Y  +359.106, Z    +0.000, E1  +320.118, E3 -347123.996}
SPL {X  -157.143, Y  +352.453, Z    +0.000, E1  +320.322, E3 -347141.927}
SPL {X  -156.148, Y  +347.650, Z    +0.000, E1  +320.549, E3 -347155.113}
SPL {X  -155.268, Y  +343.918, Z    +0.000, E1  +320.696, E3 -347165.394}
SPL {X  -153.936, Y  +338.906, Z    +0.000, E1  +320.911, E3 -347179.333}
SPL {X  -152.628, Y  +334.526, Z    +0.000, E1  +321.188, E3 -347191.736}
SPL {X  -151.010, Y  +329.654, Z    +0.000, E1  +326.674, E3 -347249.571}
ENDSPLINE

SPLINE
SPL {X  -157.513, Y  +354.453, Z    +0.000, E1  +340.941, E3 -347295.606}
SPL {X  -159.408, Y  +368.861, Z    +0.000, E1  +348.865, E3 -347305.029}
SPL {X  -159.941, Y  +378.532, Z    +0.000, E1  +354.551, E3 -347308.634}
SPL {X  -159.990, Y  +383.966, Z    +0.000, E1  +358.149, E3 -347310.086}
SPL {X  -159.990, Y  +388.001, Z    +0.000, E1  +361.086, E3 -347311.021}
SPL {X  -159.990, Y  +392.647, Z    +0.000, E1  +364.974, E3 -347312.160}
SPL {X  -159.990, Y  +397.943, Z    +0.000, E1  +369.963, E3 -347313.744}
SPL {X  -159.990, Y  +407.689, Z    +0.000, E1  +378.860, E3 -347318.399}
SPL {X  -159.990, Y  +434.822, Z    +0.000, E1  +394.625, E3 -347342.943}
SPL {X  -159.990, Y  +460.330, Z    +0.000, E1  +398.908, E3 -347387.218}
SPL {X  -159.990, Y  +464.953, Z    +0.000, E1  +398.907, E3 -347399.376}
SPL {X  -159.990, Y  +469.353, Z    +0.000, E1  +398.902, E3 -347410.957}
SPL {X  -159.990, Y  +475.034, Z    +0.000, E1  +398.936, E3 -347425.872}
SPL {X  -159.990, Y  +481.308, Z    +0.000, E1  +398.917, E3 -347442.383}
SPL {X  -159.990, Y  +485.396, Z    +0.000, E1  +398.893, E3 -347453.142}
SPL {X  -159.990, Y  +488.362, Z    +0.000, E1  +398.896, E3 -347460.926}
SPL {X  -159.990, Y  +492.629, Z    +0.000, E1  +398.922, E3 -347472.097}
SPL {X  -159.990, Y  +497.431, Z    +0.000, E1  +398.905, E3 -347484.763}
SPL {X  -159.990, Y  +502.093, Z    +0.000, E1  +398.909, E3 -347497.038}
SPL {X  -159.990, Y  +507.821, Z    +0.000, E1  +398.930, E3 -347512.058}
SPL {X  -159.990, Y  +513.533, Z    +0.000, E1  +398.910, E3 -347527.117}
SPL {X  -159.990, Y  +519.462, Z    +0.000, E1  +398.933, E3 -347542.670}
SPL {X  -159.990, Y  +524.415, Z    +0.000, E1  +398.896, E3 -347555.734}
SPL {X  -159.990, Y  +528.627, Z    +0.000, E1  +398.910, E3 -347566.795}
SPL {X  -159.990, Y  +533.053, Z    +0.000, E1  +398.899, E3 -347578.452}
SPL {X  -159.990, Y  +537.174, Z    +0.000, E1  +398.910, E3 -347589.267}
SPL {X  -159.990, Y  +541.259, Z    +0.000, E1  +398.888, E3 -347600.066}
SPL {X  -159.990, Y  +545.676, Z    +0.000, E1  +398.913, E3 -347611.637}
SPL {X  -159.990, Y  +550.777, Z    +0.000, E1  +398.906, E3 -347625.056}
SPL {X  -159.990, Y  +554.638, Z    +0.000, E1  +398.890, E3 -347635.227}
SPL {X  -159.990, Y  +557.678, Z    +0.000, E1  +398.893, E3 -347643.203}
SPL {X  -159.990, Y  +561.696, Z    +0.000, E1  +398.912, E3 -347653.728}
SPL {X  -159.990, Y  +566.650, Z    +0.000, E1  +398.917, E3 -347666.742}
SPL {X  -159.990, Y  +571.814, Z    +0.000, E1  +398.914, E3 -347680.345}
SPL {X  -159.990, Y  +577.636, Z    +0.000, E1  +398.929, E3 -347695.642}
SPL {X  -159.990, Y  +583.167, Z    +0.000, E1  +398.906, E3 -347710.217}
SPL {X  -159.990, Y  +589.106, Z    +0.000, E1  +398.939, E3 -347725.785}
SPL {X  -159.990, Y  +594.201, Z    +0.000, E1  +398.894, E3 -347739.253}
SPL {X  -159.990, Y  +599.478, Z    +0.000, E1  +398.941, E3 -347753.057}
SPL {X  -159.990, Y  +606.904, Z    +0.000, E1  +398.953, E3 -347772.570}
SPL {X  -159.990, Y  +614.125, Z    +0.000, E1  +398.936, E3 -347791.582}
SPL {X  -159.990, Y  +619.061, Z    +0.000, E1  +398.894, E3 -347804.614}
SPL {X  -159.990, Y  +623.264, Z    +0.000, E1  +398.906, E3 -347815.663}
SPL {X  -159.990, Y  +628.669, Z    +0.000, E1  +398.928, E3 -347829.831}
SPL {X  -159.990, Y  +634.089, Z    +0.000, E1  +398.907, E3 -347844.107}
SPL {X  -159.990, Y  +638.639, Z    +0.000, E1  +398.904, E3 -347856.092}
SPL {X  -159.990, Y  +643.555, Z    +0.000, E1  +398.910, E3 -347869.012}
SPL {X  -159.990, Y  +649.380, Z    +0.000, E1  +398.930, E3 -347884.290}
SPL {X  -159.990, Y  +654.813, Z    +0.000, E1  +398.905, E3 -347898.614}
SPL {X  -159.990, Y  +658.715, Z    +0.000, E1  +398.892, E3 -347908.895}
SPL {X  -159.990, Y  +661.848, Z    +0.000, E1  +398.892, E3 -347917.134}
SPL {X  -159.990, Y  +665.703, Z    +0.000, E1  +398.903, E3 -347927.253}
SPL {X  -159.990, Y  +669.966, Z    +0.000, E1  +398.902, E3 -347938.460}
SPL {X  -159.954, Y  +674.895, Z    +0.000, E1  +398.910, E3 -347951.439}
SPL {X  -159.761, Y  +680.061, Z    +0.000, E1  +398.873, E3 -347965.218}
SPL {X  -159.443, Y  +684.716, Z    +0.000, E1  +398.815, E3 -347977.784}
SPL {X  -158.962, Y  +689.604, Z    +0.000, E1  +398.740, E3 -347991.153}
SPL {X  -158.318, Y  +694.567, Z    +0.000, E1  +398.614, E3 -348004.914}
SPL {X  -157.472, Y  +699.775, Z    +0.000, E1  +398.483, E3 -348019.474}
SPL {X  -156.506, Y  +704.705, Z    +0.000, E1  +398.294, E3 -348033.474}
SPL {X  -155.680, Y  +708.387, Z    +0.000, E1  +398.127, E3 -348044.045}
SPL {X  -154.586, Y  +712.730, Z    +0.000, E1  +397.967, E3 -348056.542}
SPL {X  -153.345, Y  +717.131, Z    +0.000, E1  +397.713, E3 -348069.426}
SPL {X  -151.080, Y  +724.146, Z    +0.000, E1  +393.201, E3 -348127.880}
ENDSPLINE

SPLINE
SPL {X  -157.921, Y  +697.149, Z    +0.000, E1  +377.701, E3 -348179.440}
SPL {X  -159.579, Y  +682.959, Z    +0.000, E1  +369.793, E3 -348187.389}
SPL {X  -159.938, Y  +675.561, Z    +0.000, E1  +365.399, E3 -348189.811}
SPL {X  -159.990, Y  +669.910, Z    +0.000, E1  +361.710, E3 -348191.102}
SPL {X  -159.990, Y  +665.465, Z    +0.000, E1  +358.378, E3 -348192.019}
SPL {X  -159.990, Y  +661.791, Z    +0.000, E1  +355.213, E3 -348192.857}
SPL {X  -159.990, Y  +656.991, Z    +0.000, E1  +350.742, E3 -348194.276}
SPL {X  -159.990, Y  +649.722, Z    +0.000, E1  +343.777, E3 -348197.195}
SPL {X  -159.990, Y  +645.752, Z    +0.000, E1  +340.157, E3 -348199.136}
SPL {X  -159.990, Y  +620.451, Z    +0.000, E1  +325.419, E3 -348221.853}
SPL {X  -159.990, Y  +591.256, Z    +0.000, E1  +319.966, E3 -348268.347}
SPL {X  -159.990, Y  +586.740, Z    +0.000, E1  +319.956, E3 -348279.737}
SPL {X  -159.990, Y  +581.814, Z    +0.000, E1  +319.956, E3 -348292.176}
SPL {X  -159.990, Y  +577.274, Z    +0.000, E1  +319.964, E3 -348303.654}
SPL {X  -159.990, Y  +572.933, Z    +0.000, E1  +319.959, E3 -348314.595}
SPL {X  -159.990, Y  +568.504, Z    +0.000, E1  +319.956, E3 -348325.758}
SPL {X  -159.990, Y  +563.189, Z    +0.000, E1  +319.932, E3 -348339.131}
SPL {X  -159.990, Y  +557.707, Z    +0.000, E1  +319.949, E3 -348352.986}
SPL {X  -159.990, Y  +552.104, Z    +0.000, E1  +319.922, E3 -348367.061}
SPL {X  -159.990, Y  +545.912, Z    +0.000, E1  +319.929, E3 -348382.711}
SPL {X  -159.990, Y  +540.054, Z    +0.000, E1  +319.939, E3 -348397.538}
SPL {X  -159.990, Y  +533.683, Z    +0.000, E1  +319.916, E3 -348413.563}
SPL {X  -159.990, Y  +527.393, Z    +0.000, E1  +319.924, E3 -348429.435}
SPL {X  -159.990, Y  +522.533, Z    +0.000, E1  +319.951, E3 -348441.733}
SPL {X  -159.990, Y  +496.806, Z    +0.000, E1  +312.216, E3 -348451.940}
SPL {X  -159.990, Y  +490.245, Z    +0.000, E1  +312.831, E3 -348468.472}
SPL {X  -159.990, Y  +486.737, Z    +0.000, E1  +313.729, E3 -348480.478}
SPL {X  -159.990, Y  +483.955, Z    +0.000, E1  +314.316, E3 -348489.770}
SPL {X  -159.990, Y  +479.762, Z    +0.000, E1  +315.381, E3 -348505.161}
SPL {X  -159.990, Y  +474.562, Z    +0.000, E1  +316.600, E3 -348523.830}
SPL {X  -159.990, Y  +470.788, Z    +0.000, E1  +317.853, E3 -348539.713}
SPL {X  -159.990, Y  +467.944, Z    +0.000, E1  +318.635, E3 -348551.035}
SPL {X  -159.990, Y  +465.057, Z    +0.000, E1  +319.375, E3 -348562.600}
SPL {X  -159.990, Y  +461.409, Z    +0.000, E1  +319.848, E3 -348574.499}
SPL {X  -159.990, Y  +456.934, Z    +0.000, E1  +319.854, E3 -348585.775}
SPL {X  -159.990, Y  +452.940, Z    +0.000, E1  +319.854, E3 -348595.820}
SPL {X  -159.990, Y  +448.856, Z    +0.000, E1  +319.859, E3 -348606.103}
SPL {X  -159.990, Y  +444.973, Z    +0.000, E1  +319.856, E3 -348615.868}
SPL {X  -159.990, Y  +439.927, Z    +0.000, E1  +319.837, E3 -348628.525}
SPL {X  -159.990, Y  +435.246, Z    +0.000, E1  +319.853, E3 -348640.334}
SPL {X  -159.990, Y  +430.690, Z    +0.000, E1  +319.854, E3 -348651.796}
SPL {X  -159.990, Y  +426.145, Z    +0.000, E1  +319.853, E3 -348663.235}
SPL {X  -159.990, Y  +421.880, Z    +0.000, E1  +319.860, E3 -348673.968}
SPL {X  -159.990, Y  +416.246, Z    +0.000, E1  +319.819, E3 -348688.097}
SPL {X  -159.990, Y  +409.936, Z    +0.000, E1  +319.849, E3 -348704.034}
SPL {X  -159.990, Y  +404.988, Z    +0.000, E1  +319.861, E3 -348716.500}
SPL {X  -159.990, Y  +400.535, Z    +0.000, E1  +319.859, E3 -348727.698}
SPL {X  -159.990, Y  +396.024, Z    +0.000, E1  +319.860, E3 -348739.054}
SPL {X  -159.990, Y  +391.614, Z    +0.000, E1  +319.860, E3 -348750.147}
SPL {X  -159.990, Y  +387.212, Z    +0.000, E1  +319.859, E3 -348761.219}
SPL {X  -159.990, Y  +382.743, Z    +0.000, E1  +319.857, E3 -348772.461}
SPL {X  -159.925, Y  +377.946, Z    +0.000, E1  +319.864, E3 -348784.598}
SPL {X  -159.703, Y  +372.915, Z    +0.000, E1  +319.904, E3 -348797.498}
SPL {X  -159.358, Y  +368.290, Z    +0.000, E1  +319.961, E3 -348809.460}
SPL {X  -158.955, Y  +364.333, Z    +0.000, E1  +320.046, E3 -348819.863}
SPL {X  -158.482, Y  +360.589, Z    +0.000, E1  +320.125, E3 -348829.789}
SPL {X  -157.729, Y  +355.695, Z    +0.000, E1  +320.237, E3 -348842.862}
SPL {X  -156.893, Y  +351.173, Z    +0.000, E1  +320.410, E3 -348855.145}
SPL {X  -156.148, Y  +347.650, Z    +0.000, E1  +320.549, E3 -348864.791}
SPL {X  -155.268, Y  +343.918, Z    +0.000, E1  +320.696, E3 -348875.072}
SPL {X  -154.153, Y  +339.677, Z    +0.000, E1  +320.896, E3 -348886.879}
SPL {X  -152.885, Y  +335.352, Z    +0.000, E1  +321.114, E3 -348899.033}
SPL {X  -151.010, Y  +329.654, Z    +0.000, E1  +326.674, E3 -348959.249}
ENDSPLINE

SPLINE
SPL {X  -157.513, Y  +354.453, Z    +0.000, E1  +340.941, E3 -349005.283}
SPL {X  -159.408, Y  +368.861, Z    +0.000, E1  +348.865, E3 -349014.706}
SPL {X  -159.941, Y  +378.532, Z    +0.000, E1  +354.551, E3 -349018.312}
SPL {X  -159.990, Y  +383.966, Z    +0.000, E1  +358.149, E3 -349019.763}
SPL {X  -159.990, Y  +389.165, Z    +0.000, E1  +361.929, E3 -349020.965}
SPL {X  -159.990, Y  +396.368, Z    +0.000, E1  +368.359, E3 -349022.937}
SPL {X  -159.990, Y  +407.689, Z    +0.000, E1  +378.860, E3 -349028.076}
SPL {X  -159.990, Y  +434.822, Z    +0.000, E1  +394.625, E3 -349052.620}
SPL {X  -159.990, Y  +460.330, Z    +0.000, E1  +398.908, E3 -349096.896}
SPL {X  -159.990, Y  +464.953, Z    +0.000, E1  +398.907, E3 -349109.054}
SPL {X  -159.990, Y  +469.353, Z    +0.000, E1  +398.902, E3 -349120.634}
SPL {X  -159.990, Y  +473.222, Z    +0.000, E1  +398.891, E3 -349130.843}
SPL {X  -159.990, Y  +477.957, Z    +0.000, E1  +398.922, E3 -349143.248}
SPL {X  -159.990, Y  +482.463, Z    +0.000, E1  +398.891, E3 -349155.136}
SPL {X  -159.990, Y  +486.996, Z    +0.000, E1  +398.928, E3 -349166.968}
SPL {X  -159.990, Y  +492.629, Z    +0.000, E1  +398.922, E3 -349181.774}
SPL {X  -159.990, Y  +497.431, Z    +0.000, E1  +398.905, E3 -349194.441}
SPL {X  -159.990, Y  +502.093, Z    +0.000, E1  +398.909, E3 -349206.715}
SPL {X  -159.990, Y  +507.821, Z    +0.000, E1  +398.930, E3 -349221.735}
SPL {X  -159.990, Y  +513.533, Z    +0.000, E1  +398.910, E3 -349236.795}
SPL {X  -159.990, Y  +518.435, Z    +0.000, E1  +398.905, E3 -349249.690}
SPL {X  -159.990, Y  +523.478, Z    +0.000, E1  +398.918, E3 -349262.918}
SPL {X  -159.990, Y  +528.627, Z    +0.000, E1  +398.910, E3 -349276.472}
SPL {X  -159.990, Y  +534.392, Z    +0.000, E1  +398.932, E3 -349291.602}
SPL {X  -159.990, Y  +540.299, Z    +0.000, E1  +398.912, E3 -349307.177}
SPL {X  -159.990, Y  +545.676, Z    +0.000, E1  +398.913, E3 -349321.314}
SPL {X  -159.990, Y  +550.777, Z    +0.000, E1  +398.906, E3 -349334.734}
SPL {X  -159.990, Y  +556.271, Z    +0.000, E1  +398.927, E3 -349349.136}
SPL {X  -159.990, Y  +561.696, Z    +0.000, E1  +398.912, E3 -349363.406}
SPL {X  -159.990, Y  +566.650, Z    +0.000, E1  +398.917, E3 -349376.419}
SPL {X  -159.990, Y  +571.814, Z    +0.000, E1  +398.914, E3 -349390.022}
SPL {X  -159.990, Y  +577.636, Z    +0.000, E1  +398.929, E3 -349405.319}
SPL {X  -159.990, Y  +583.167, Z    +0.000, E1  +398.906, E3 -349419.895}
SPL {X  -159.990, Y  +589.106, Z    +0.000, E1  +398.939, E3 -349435.462}
SPL {X  -159.990, Y  +596.185, Z    +0.000, E1  +398.945, E3 -349454.071}
SPL {X  -159.990, Y  +602.727, Z    +0.000, E1  +398.920, E3 -349471.310}
SPL {X  -159.990, Y  +608.112, Z    +0.000, E1  +398.911, E3 -349485.485}
SPL {X  -159.990, Y  +614.125, Z    +0.000, E1  +398.936, E3 -349501.260}
SPL {X  -159.990, Y  +619.061, Z    +0.000, E1  +398.894, E3 -349514.291}
SPL {X  -159.990, Y  +623.264, Z    +0.000, E1  +398.906, E3 -349525.340}
SPL {X  -159.990, Y  +628.669, Z    +0.000, E1  +398.928, E3 -349539.508}
SPL {X  -159.990, Y  +634.089, Z    +0.000, E1  +398.907, E3 -349553.784}
SPL {X  -159.990, Y  +638.639, Z    +0.000, E1  +398.904, E3 -349565.770}
SPL {X  -159.990, Y  +644.750, Z    +0.000, E1  +398.946, E3 -349581.775}
SPL {X  -159.990, Y  +650.458, Z    +0.000, E1  +398.900, E3 -349596.848}
SPL {X  -159.990, Y  +654.813, Z    +0.000, E1  +398.905, E3 -349608.292}
SPL {X  -159.990, Y  +660.353, Z    +0.000, E1  +398.930, E3 -349622.823}
SPL {X  -159.990, Y  +665.703, Z    +0.000, E1  +398.903, E3 -349636.930}
SPL {X  -159.990, Y  +671.472, Z    +0.000, E1  +398.942, E3 -349652.035}
SPL {X  -159.920, Y  +676.216, Z    +0.000, E1  +398.875, E3 -349664.670}
SPL {X  -159.761, Y  +680.061, Z    +0.000, E1  +398.873, E3 -349674.896}
SPL {X  -159.443, Y  +684.716, Z    +0.000, E1  +398.815, E3 -349687.461}
SPL {X  -158.962, Y  +689.604, Z    +0.000, E1  +398.740, E3 -349700.830}
SPL {X  -158.318, Y  +694.567, Z    +0.000, E1  +398.614, E3 -349714.591}
SPL {X  -157.472, Y  +699.775, Z    +0.000, E1  +398.483, E3 -349729.151}
SPL {X  -156.506, Y  +704.705, Z    +0.000, E1  +398.294, E3 -349743.151}
SPL {X  -155.357, Y  +709.721, Z    +0.000, E1  +398.108, E3 -349757.506}
SPL {X  -154.005, Y  +714.851, Z    +0.000, E1  +397.854, E3 -349772.401}
SPL {X  -153.100, Y  +717.944, Z    +0.000, E1  +397.652, E3 -349781.511}
SPL {X  -151.080, Y  +724.146, Z    +0.000, E1  +393.201, E3 -349837.557}
ENDSPLINE

SPLINE
SPL {X  -157.921, Y  +697.149, Z    +0.000, E1  +377.701, E3 -349889.118}
SPL {X  -159.579, Y  +682.959, Z    +0.000, E1  +369.793, E3 -349897.066}
SPL {X  -159.938, Y  +675.561, Z    +0.000, E1  +365.399, E3 -349899.488}
SPL {X  -159.990, Y  +669.910, Z    +0.000, E1  +361.710, E3 -349900.779}
SPL {X  -159.990, Y  +665.465, Z    +0.000, E1  +358.378, E3 -349901.697}
SPL {X  -159.990, Y  +661.791, Z    +0.000, E1  +355.213, E3 -349902.534}
SPL {X  -159.990, Y  +656.991, Z    +0.000, E1  +350.742, E3 -349903.954}
SPL {X  -159.990, Y  +649.722, Z    +0.000, E1  +343.777, E3 -349906.872}
SPL {X  -159.990, Y  +645.752, Z    +0.000, E1  +340.157, E3 -349908.813}
SPL {X  -159.990, Y  +620.451, Z    +0.000, E1  +325.419, E3 -349931.530}
SPL {X  -159.990, Y  +591.256, Z    +0.000, E1  +319.966, E3 -349978.024}
SPL {X  -159.990, Y  +586.740, Z    +0.000, E1  +319.956, E3 -349989.414}
SPL {X  -159.990, Y  +581.814, Z    +0.000, E1  +319.956, E3 -350001.854}
SPL {X  -159.990, Y  +577.274, Z    +0.000, E1  +319.964, E3 -350013.331}
SPL {X  -159.990, Y  +572.933, Z    +0.000, E1  +319.959, E3 -350024.272}
SPL {X  -159.990, Y  +568.504, Z    +0.000, E1  +319.956, E3 -350035.435}
SPL {X  -159.990, Y  +563.189, Z    +0.000, E1  +319.932, E3 -350048.809}
SPL {X  -159.990, Y  +557.707, Z    +0.000, E1  +319.949, E3 -350062.664}
SPL {X  -159.990, Y  +552.104, Z    +0.000, E1  +319.922, E3 -350076.739}
SPL {X  -159.990, Y  +545.912, Z    +0.000, E1  +319.929, E3 -350092.388}
SPL {X  -159.990, Y  +540.054, Z    +0.000, E1  +319.939, E3 -350107.215}
SPL {X  -159.990, Y  +533.683, Z    +0.000, E1  +319.916, E3 -350123.240}
SPL {X  -159.990, Y  +527.393, Z    +0.000, E1  +319.924, E3 -350139.113}
SPL {X  -159.990, Y  +522.533, Z    +0.000, E1  +319.951, E3 -350151.410}
SPL {X  -159.990, Y  +502.378, Z    +0.000, E1  +313.079, E3 -350155.814}
SPL {X  -159.990, Y  +493.568, Z    +0.000, E1  +312.053, E3 -350166.982}
SPL {X  -159.990, Y  +488.437, Z    +0.000, E1  +313.241, E3 -350184.197}
SPL {X  -159.990, Y  +483.955, Z    +0.000, E1  +314.316, E3 -350199.447}
SPL {X  -159.990, Y  +480.580, Z    +0.000, E1  +315.242, E3 -350212.068}
SPL {X  -159.990, Y  +476.546, Z    +0.000, E1  +316.165, E3 -350226.363}
SPL {X  -159.990, Y  +472.671, Z    +0.000, E1  +317.192, E3 -350241.190}
SPL {X  -159.990, Y  +468.809, Z    +0.000, E1  +318.343, E3 -350257.119}
SPL {X  -159.990, Y  +465.057, Z    +0.000, E1  +319.375, E3 -350272.277}
SPL {X  -159.990, Y  +461.409, Z    +0.000, E1  +319.848, E3 -350284.177}
SPL {X  -159.990, Y  +456.934, Z    +0.000, E1  +319.854, E3 -350295.452}
SPL {X  -159.990, Y  +452.940, Z    +0.000, E1  +319.854, E3 -350305.497}
SPL {X  -159.990, Y  +448.856, Z    +0.000, E1  +319.859, E3 -350315.780}
SPL {X  -159.990, Y  +443.741, Z    +0.000, E1  +319.827, E3 -350328.598}
SPL {X  -159.990, Y  +436.703, Z    +0.000, E1  +319.809, E3 -350346.280}
SPL {X  -159.990, Y  +430.690, Z    +0.000, E1  +319.854, E3 -350361.473}
SPL {X  -159.990, Y  +426.145, Z    +0.000, E1  +319.853, E3 -350372.913}
SPL {X  -159.990, Y  +421.880, Z    +0.000, E1  +319.860, E3 -350383.646}
SPL {X  -159.990, Y  +417.572, Z    +0.000, E1  +319.852, E3 -350394.473}
SPL {X  -159.990, Y  +412.619, Z    +0.000, E1  +319.850, E3 -350406.964}
SPL {X  -159.990, Y  +406.264, Z    +0.000, E1  +319.825, E3 -350422.912}
SPL {X  -159.990, Y  +400.535, Z    +0.000, E1  +319.859, E3 -350437.375}
SPL {X  -159.990, Y  +396.024, Z    +0.000, E1  +319.860, E3 -350448.731}
SPL {X  -159.990, Y  +391.614, Z    +0.000, E1  +319.860, E3 -350459.825}
SPL {X  -159.990, Y  +387.212, Z    +0.000, E1  +319.859, E3 -350470.897}
SPL {X  -159.990, Y  +382.743, Z    +0.000, E1  +319.857, E3 -350482.138}
SPL {X  -159.925, Y  +377.946, Z    +0.000, E1  +319.864, E3 -350494.275}
SPL {X  -159.703, Y  +372.915, Z    +0.000, E1  +319.904, E3 -350507.175}
SPL {X  -159.358, Y  +368.290, Z    +0.000, E1  +319.961, E3 -350519.138}
SPL {X  -158.955, Y  +364.333, Z    +0.000, E1  +320.046, E3 -350529.540}
SPL {X  -158.482, Y  +360.589, Z    +0.000, E1  +320.125, E3 -350539.466}
SPL {X  -157.729, Y  +355.695, Z    +0.000, E1  +320.237, E3 -350552.539}
SPL {X  -156.893, Y  +351.173, Z    +0.000, E1  +320.410, E3 -350564.822}
SPL {X  -156.148, Y  +347.650, Z    +0.000, E1  +320.549, E3 -350574.468}
SPL {X  -155.268, Y  +343.918, Z    +0.000, E1  +320.696, E3 -350584.749}
SPL {X  -154.153, Y  +339.677, Z    +0.000, E1  +320.896, E3 -350596.556}
SPL {X  -152.885, Y  +335.352, Z    +0.000, E1  +321.114, E3 -350608.710}
SPL {X  -151.010, Y  +329.654, Z    +0.000, E1  +326.674, E3 -350668.926}
ENDSPLINE

SPLINE
SPL {X  -157.513, Y  +354.453, Z    +0.000, E1  +340.941, E3 -350714.961}
SPL {X  -159.638, Y  +371.886, Z    +0.000, E1  +350.545, E3 -350725.623}
SPL {X  -159.990, Y  +382.357, Z    +0.000, E1  +356.972, E3 -350729.038}
SPL {X  -159.990, Y  +389.165, Z    +0.000, E1  +361.929, E3 -350730.643}
SPL {X  -159.990, Y  +396.368, Z    +0.000, E1  +368.359, E3 -350732.615}
SPL {X  -159.990, Y  +407.689, Z    +0.000, E1  +378.860, E3 -350737.754}
SPL {X  -159.990, Y  +434.822, Z    +0.000, E1  +394.625, E3 -350762.298}
SPL {X  -159.990, Y  +460.330, Z    +0.000, E1  +398.908, E3 -350806.573}
SPL {X  -159.990, Y  +464.953, Z    +0.000, E1  +398.907, E3 -350818.731}
SPL {X  -159.990, Y  +469.353, Z    +0.000, E1  +398.902, E3 -350830.312}
SPL {X  -159.990, Y  +475.034, Z    +0.000, E1  +398.936, E3 -350845.227}
SPL {X  -159.990, Y  +481.308, Z    +0.000, E1  +398.917, E3 -350861.737}
SPL {X  -159.990, Y  +485.396, Z    +0.000, E1  +398.893, E3 -350872.497}
SPL {X  -159.990, Y  +488.362, Z    +0.000, E1  +398.896, E3 -350880.280}
SPL {X  -159.990, Y  +492.629, Z    +0.000, E1  +398.922, E3 -350891.452}
SPL {X  -159.990, Y  +497.431, Z    +0.000, E1  +398.905, E3 -350904.118}
SPL {X  -159.990, Y  +502.093, Z    +0.000, E1  +398.909, E3 -350916.393}
SPL {X  -159.990, Y  +507.821, Z    +0.000, E1  +398.930, E3 -350931.413}
SPL {X  -159.990, Y  +513.533, Z    +0.000, E1  +398.910, E3 -350946.472}
SPL {X  -159.990, Y  +518.435, Z    +0.000, E1  +398.905, E3 -350959.367}
SPL {X  -159.990, Y  +523.478, Z    +0.000, E1  +398.918, E3 -350972.596}
SPL {X  -159.990, Y  +528.627, Z    +0.000, E1  +398.910, E3 -350986.149}
SPL {X  -159.990, Y  +533.053, Z    +0.000, E1  +398.899, E3 -350997.807}
SPL {X  -159.990, Y  +537.174, Z    +0.000, E1  +398.910, E3 -351008.621}
SPL {X  -159.990, Y  +541.259, Z    +0.000, E1  +398.888, E3 -351019.421}
SPL {X  -159.990, Y  +545.676, Z    +0.000, E1  +398.913, E3 -351030.992}
SPL {X  -159.990, Y  +550.777, Z    +0.000, E1  +398.906, E3 -351044.411}
SPL {X  -159.990, Y  +554.638, Z    +0.000, E1  +398.890, E3 -351054.582}
SPL {X  -159.990, Y  +557.678, Z    +0.000, E1  +398.893, E3 -351062.558}
SPL {X  -159.990, Y  +561.696, Z    +0.000, E1  +398.912, E3 -351073.083}
SPL {X  -159.990, Y  +566.650, Z    +0.000, E1  +398.917, E3 -351086.097}
SPL {X  -159.990, Y  +571.814, Z    +0.000, E1  +398.914, E3 -351099.699}
SPL {X  -159.990, Y  +577.636, Z    +0.000, E1  +398.929, E3 -351114.997}
SPL {X  -159.990, Y  +583.167, Z    +0.000, E1  +398.906, E3 -351129.572}
SPL {X  -159.990, Y  +587.761, Z    +0.000, E1  +398.902, E3 -351141.657}
SPL {X  -159.990, Y  +592.962, Z    +0.000, E1  +398.925, E3 -351155.301}
SPL {X  -159.990, Y  +597.767, Z    +0.000, E1  +398.897, E3 -351167.977}
SPL {X  -159.990, Y  +602.727, Z    +0.000, E1  +398.920, E3 -351180.988}
SPL {X  -159.990, Y  +608.112, Z    +0.000, E1  +398.911, E3 -351195.162}
SPL {X  -159.990, Y  +614.125, Z    +0.000, E1  +398.936, E3 -351210.937}
SPL {X  -159.990, Y  +619.061, Z    +0.000, E1  +398.894, E3 -351223.969}
SPL {X  -159.990, Y  +623.264, Z    +0.000, E1  +398.906, E3 -351235.018}
SPL {X  -159.990, Y  +628.669, Z    +0.000, E1  +398.928, E3 -351249.186}
SPL {X  -159.990, Y  +634.089, Z    +0.000, E1  +398.907, E3 -351263.462}
SPL {X  -159.990, Y  +638.639, Z    +0.000, E1  +398.904, E3 -351275.447}
SPL {X  -159.990, Y  +643.555, Z    +0.000, E1  +398.910, E3 -351288.367}
SPL {X  -159.990, Y  +649.380, Z    +0.000, E1  +398.930, E3 -351303.645}
SPL {X  -159.990, Y  +654.813, Z    +0.000, E1  +398.905, E3 -351317.969}
SPL {X  -159.990, Y  +660.353, Z    +0.000, E1  +398.930, E3 -351332.501}
SPL {X  -159.990, Y  +665.703, Z    +0.000, E1  +398.903, E3 -351346.608}
SPL {X  -159.990, Y  +671.472, Z    +0.000, E1  +398.942, E3 -351361.712}
SPL {X  -159.920, Y  +676.216, Z    +0.000, E1  +398.875, E3 -351374.348}
SPL {X  -159.761, Y  +680.061, Z    +0.000, E1  +398.873, E3 -351384.573}
SPL {X  -159.443, Y  +684.716, Z    +0.000, E1  +398.815, E3 -351397.138}
SPL {X  -158.962, Y  +689.604, Z    +0.000, E1  +398.740, E3 -351410.508}
SPL {X  -158.318, Y  +694.567, Z    +0.000, E1  +398.614, E3 -351424.269}
SPL {X  -157.472, Y  +699.775, Z    +0.000, E1  +398.483, E3 -351438.828}
SPL {X  -156.506, Y  +704.705, Z    +0.000, E1  +398.294, E3 -351452.829}
SPL {X  -155.357, Y  +709.721, Z    +0.000, E1  +398.108, E3 -351467.184}
SPL {X  -154.286, Y  +713.838, Z    +0.000, E1  +397.877, E3 -351479.167}
SPL {X  -153.345, Y  +717.131, Z    +0.000, E1  +397.713, E3 -351488.781}
SPL {X  -151.080, Y  +724.146, Z    +0.000, E1  +393.201, E3 -351547.234}
ENDSPLINE

SPLINE
SPL {X  -157.921, Y  +697.149, Z    +0.000, E1  +377.701, E3 -351598.795}
SPL {X  -159.579, Y  +682.959, Z    +0.000, E1  +369.793, E3 -351606.744}
SPL {X  -159.938, Y  +675.561, Z    +0.000, E1  +365.399, E3 -351609.166}
SPL {X  -159.990, Y  +669.910, Z    +0.000, E1  +361.710, E3 -351610.457}
SPL {X  -159.990, Y  +665.465, Z    +0.000, E1  +358.378, E3 -351611.374}
SPL {X  -159.990, Y  +661.791, Z    +0.000, E1  +355.213, E3 -351612.212}
SPL {X  -159.990, Y  +656.991, Z    +0.000, E1  +350.742, E3 -351613.631}
SPL {X  -159.990, Y  +648.067, Z    +0.000, E1  +342.328, E3 -351617.361}
SPL {X  -159.990, Y  +620.451, Z    +0.000, E1  +325.419, E3 -351641.208}
SPL {X  -159.990, Y  +591.256, Z    +0.000, E1  +319.966, E3 -351687.701}
SPL {X  -159.990, Y  +586.740, Z    +0.000, E1  +319.956, E3 -351699.092}
SPL {X  -159.990, Y  +581.814, Z    +0.000, E1  +319.956, E3 -351711.531}
SPL {X  -159.990, Y  +577.274, Z    +0.000, E1  +319.964, E3 -351723.009}
SPL {X  -159.990, Y  +572.933, Z    +0.000, E1  +319.959, E3 -351733.950}
SPL {X  -159.990, Y  +568.504, Z    +0.000, E1  +319.956, E3 -351745.112}
SPL {X  -159.990, Y  +563.189, Z    +0.000, E1  +319.932, E3 -351758.486}
SPL {X  -159.990, Y  +557.707, Z    +0.000, E1  +319.949, E3 -351772.341}
SPL {X  -159.990, Y  +553.571, Z    +0.000, E1  +319.954, E3 -351782.760}
SPL {X  -159.990, Y  +549.413, Z    +0.000, E1  +319.938, E3 -351793.226}
SPL {X  -159.990, Y  +543.439, Z    +0.000, E1  +319.921, E3 -351808.314}
SPL {X  -159.990, Y  +537.213, Z    +0.000, E1  +319.937, E3 -351824.056}
SPL {X  -159.990, Y  +532.291, Z    +0.000, E1  +319.951, E3 -351836.481}
SPL {X  -159.990, Y  +527.393, Z    +0.000, E1  +319.924, E3 -351848.790}
SPL {X  -159.990, Y  +522.533, Z    +0.000, E1  +319.951, E3 -351861.088}
SPL {X  -159.990, Y  +496.806, Z    +0.000, E1  +312.216, E3 -351871.295}
SPL {X  -159.990, Y  +490.245, Z    +0.000, E1  +312.831, E3 -351887.827}
SPL {X  -159.990, Y  +486.737, Z    +0.000, E1  +313.729, E3 -351899.833}
SPL {X  -159.990, Y  +483.955, Z    +0.000, E1  +314.316, E3 -351909.125}
SPL {X  -159.990, Y  +480.580, Z    +0.000, E1  +315.242, E3 -351921.746}
SPL {X  -159.990, Y  +476.546, Z    +0.000, E1  +316.165, E3 -351936.040}
SPL {X  -159.990, Y  +473.377, Z    +0.000, E1  +316.953, E3 -351947.655}
SPL {X  -159.990, Y  +470.788, Z    +0.000, E1  +317.853, E3 -351959.068}
SPL {X  -159.990, Y  +467.944, Z    +0.000, E1  +318.635, E3 -351970.389}
SPL {X  -159.990, Y  +465.057, Z    +0.000, E1  +319.375, E3 -351981.955}
SPL {X  -159.990, Y  +461.409, Z    +0.000, E1  +319.848, E3 -351993.854}
SPL {X  -159.990, Y  +456.934, Z    +0.000, E1  +319.854, E3 -352005.130}
SPL {X  -159.990, Y  +452.940, Z    +0.000, E1  +319.854, E3 -352015.174}
SPL {X  -159.990, Y  +448.856, Z    +0.000, E1  +319.859, E3 -352025.458}
SPL {X  -159.990, Y  +443.741, Z    +0.000, E1  +319.827, E3 -352038.276}
SPL {X  -159.990, Y  +436.703, Z    +0.000, E1  +319.809, E3 -352055.957}
SPL {X  -159.990, Y  +430.690, Z    +0.000, E1  +319.854, E3 -352071.151}
SPL {X  -159.990, Y  +426.145, Z    +0.000, E1  +319.853, E3 -352082.590}
SPL {X  -159.990, Y  +421.880, Z    +0.000, E1  +319.860, E3 -352093.323}
SPL {X  -159.990, Y  +416.246, Z    +0.000, E1  +319.819, E3 -352107.452}
SPL {X  -159.990, Y  +409.936, Z    +0.000, E1  +319.849, E3 -352123.389}
SPL {X  -159.990, Y  +404.988, Z    +0.000, E1  +319.861, E3 -352135.854}
SPL {X  -159.990, Y  +400.535, Z    +0.000, E1  +319.859, E3 -352147.052}
SPL {X  -159.990, Y  +396.024, Z    +0.000, E1  +319.860, E3 -352158.408}
SPL {X  -159.990, Y  +391.614, Z    +0.000, E1  +319.860, E3 -352169.502}
SPL {X  -159.990, Y  +387.212, Z    +0.000, E1  +319.859, E3 -352180.574}
SPL {X  -159.990, Y  +382.743, Z    +0.000, E1  +319.857, E3 -352191.816}
SPL {X  -159.925, Y  +377.946, Z    +0.000, E1  +319.864, E3 -352203.953}
SPL {X  -159.703, Y  +372.915, Z    +0.000, E1  +319.904, E3 -352216.853}
SPL {X  -159.358, Y  +368.290, Z    +0.000, E1  +319.961, E3 -352228.815}
SPL {X  -158.955, Y  +364.333, Z    +0.000, E1  +320.046, E3 -352239.218}
SPL {X  -158.482, Y  +360.589, Z    +0.000, E1  +320.125, E3 -352249.144}
SPL {X  -157.729, Y  +355.695, Z    +0.000, E1  +320.237, E3 -352262.216}
SPL {X  -156.893, Y  +351.173, Z    +0.000, E1  +320.410, E3 -352274.500}
SPL {X  -156.148, Y  +347.650, Z    +0.000, E1  +320.549, E3 -352284.146}
SPL {X  -155.268, Y  +343.918, Z    +0.000, E1  +320.696, E3 -352294.426}
SPL {X  -153.936, Y  +338.906, Z    +0.000, E1  +320.911, E3 -352308.366}
SPL {X  -152.628, Y  +334.526, Z    +0.000, E1  +321.188, E3 -352320.768}
SPL {X  -151.010, Y  +329.654, Z    +0.000, E1  +326.674, E3 -352378.604}
ENDSPLINE

SPLINE
SPL {X  -157.513, Y  +354.453, Z    +0.000, E1  +340.941, E3 -352424.638}
SPL {X  -159.408, Y  +368.861, Z    +0.000, E1  +348.865, E3 -352434.061}
SPL {X  -159.941, Y  +378.532, Z    +0.000, E1  +354.551, E3 -352437.666}
SPL {X  -159.990, Y  +383.966, Z    +0.000, E1  +358.149, E3 -352439.118}
SPL {X  -159.990, Y  +388.001, Z    +0.000, E1  +361.086, E3 -352440.053}
SPL {X  -159.990, Y  +392.647, Z    +0.000, E1  +364.974, E3 -352441.192}
SPL {X  -159.990, Y  +397.943, Z    +0.000, E1  +369.963, E3 -352442.777}
SPL {X  -159.990, Y  +406.530, Z    +0.000, E1  +377.917, E3 -352446.674}
SPL {X  -159.990, Y  +429.014, Z    +0.000, E1  +392.438, E3 -352465.331}
SPL {X  -159.990, Y  +437.635, Z    +0.000, E1  +395.495, E3 -352475.563}
SPL {X  -159.990, Y  +460.330, Z    +0.000, E1  +398.908, E3 -352516.250}
SPL {X  -159.990, Y  +464.953, Z    +0.000, E1  +398.907, E3 -352528.409}
SPL {X  -159.990, Y  +469.353, Z    +0.000, E1  +398.902, E3 -352539.989}
SPL {X  -159.990, Y  +475.034, Z    +0.000, E1  +398.936, E3 -352554.904}
SPL {X  -159.990, Y  +481.308, Z    +0.000, E1  +398.917, E3 -352571.415}
SPL {X  -159.990, Y  +485.396, Z    +0.000, E1  +398.893, E3 -352582.174}
SPL {X  -159.990, Y  +488.362, Z    +0.000, E1  +398.896, E3 -352589.958}
SPL {X  -159.990, Y  +492.629, Z    +0.000, E1  +398.922, E3 -352601.129}
SPL {X  -159.990, Y  +497.431, Z    +0.000, E1  +398.905, E3 -352613.795}
SPL {X  -159.990, Y  +502.093, Z    +0.000, E1  +398.909, E3 -352626.070}
SPL {X  -159.990, Y  +507.821, Z    +0.000, E1  +398.930, E3 -352641.090}
SPL {X  -159.990, Y  +513.533, Z    +0.000, E1  +398.910, E3 -352656.150}
SPL {X  -159.990, Y  +518.435, Z    +0.000, E1  +398.905, E3 -352669.045}
SPL {X  -159.990, Y  +523.478, Z    +0.000, E1  +398.918, E3 -352682.273}
SPL {X  -159.990, Y  +528.627, Z    +0.000, E1  +398.910, E3 -352695.827}
SPL {X  -159.990, Y  +533.053, Z    +0.000, E1  +398.899, E3 -352707.485}
SPL {X  -159.990, Y  +537.174, Z    +0.000, E1  +398.910, E3 -352718.299}
SPL {X  -159.990, Y  +541.259, Z    +0.000, E1  +398.888, E3 -352729.099}
SPL {X  -159.990, Y  +545.676, Z    +0.000, E1  +398.913, E3 -352740.669}
SPL {X  -159.990, Y  +550.777, Z    +0.000, E1  +398.906, E3 -352754.088}
SPL {X  -159.990, Y  +556.271, Z    +0.000, E1  +398.927, E3 -352768.491}
SPL {X  -159.990, Y  +561.696, Z    +0.000, E1  +398.912, E3 -352782.760}
SPL {X  -159.990, Y  +566.650, Z    +0.000, E1  +398.917, E3 -352795.774}
SPL {X  -159.990, Y  +571.814, Z    +0.000, E1  +398.914, E3 -352809.377}
SPL {X  -159.990, Y  +577.636, Z    +0.000, E1  +398.929, E3 -352824.674}
SPL {X  -159.990, Y  +583.167, Z    +0.000, E1  +398.906, E3 -352839.250}
SPL {X  -159.990, Y  +589.106, Z    +0.000, E1  +398.939, E3 -352854.817}
SPL {X  -159.990, Y  +596.185, Z    +0.000, E1  +398.945, E3 -352873.426}
SPL {X  -159.990, Y  +602.727, Z    +0.000, E1  +398.920, E3 -352890.665}
SPL {X  -159.990, Y  +608.112, Z    +0.000, E1  +398.911, E3 -352904.839}
SPL {X  -159.990, Y  +614.125, Z    +0.000, E1  +398.936, E3 -352920.614}
SPL {X  -159.990, Y  +619.061, Z    +0.000, E1  +398.894, E3 -352933.646}
SPL {X  -159.990, Y  +623.264, Z    +0.000, E1  +398.906, E3 -352944.695}
SPL {X  -159.990, Y  +628.669, Z    +0.000, E1  +398.928, E3 -352958.863}
SPL {X  -159.990, Y  +634.089, Z    +0.000, E1  +398.907, E3 -352973.139}
SPL {X  -159.990, Y  +638.639, Z    +0.000, E1  +398.904, E3 -352985.125}
SPL {X  -159.990, Y  +644.750, Z    +0.000, E1  +398.946, E3 -353001.130}
SPL {X  -159.990, Y  +650.458, Z    +0.000, E1  +398.900, E3 -353016.202}
SPL {X  -159.990, Y  +654.813, Z    +0.000, E1  +398.905, E3 -353027.647}
SPL {X  -159.990, Y  +660.353, Z    +0.000, E1  +398.930, E3 -353042.178}
SPL {X  -159.990, Y  +665.703, Z    +0.000, E1  +398.903, E3 -353056.285}
SPL {X  -159.990, Y  +671.472, Z    +0.000, E1  +398.942, E3 -353071.390}
SPL {X  -159.920, Y  +676.216, Z    +0.000, E1  +398.875, E3 -353084.025}
SPL {X  -159.761, Y  +680.061, Z    +0.000, E1  +398.873, E3 -353094.251}
SPL {X  -159.443, Y  +684.716, Z    +0.000, E1  +398.815, E3 -353106.816}
SPL {X  -158.962, Y  +689.604, Z    +0.000, E1  +398.740, E3 -353120.185}
SPL {X  -158.139, Y  +695.766, Z    +0.000, E1  +398.623, E3 -353137.231}
SPL {X  -157.275, Y  +700.848, Z    +0.000, E1  +398.415, E3 -353151.583}
SPL {X  -156.506, Y  +704.705, Z    +0.000, E1  +398.294, E3 -353162.506}
SPL {X  -155.357, Y  +709.721, Z    +0.000, E1  +398.108, E3 -353176.861}
SPL {X  -154.286, Y  +713.838, Z    +0.000, E1  +397.877, E3 -353188.844}
SPL {X  -153.345, Y  +717.131, Z    +0.000, E1  +397.713, E3 -353198.458}
SPL {X  -151.080, Y  +724.146, Z    +0.000, E1  +393.201, E3 -353256.912}
ENDSPLINE

SPLINE
SPL {X  -157.921, Y  +697.149, Z    +0.000, E1  +377.701, E3 -353308.473}
SPL {X  -159.579, Y  +682.959, Z    +0.000, E1  +369.793, E3 -353316.421}
SPL {X  -159.938, Y  +675.561, Z    +0.000, E1  +365.399, E3 -353318.843}
SPL {X  -159.990, Y  +669.910, Z    +0.000, E1  +361.710, E3 -353320.134}
SPL {X  -159.990, Y  +665.465, Z    +0.000, E1  +358.378, E3 -353321.052}
SPL {X  -159.990, Y  +661.791, Z    +0.000, E1  +355.213, E3 -353321.889}
SPL {X  -159.990, Y  +656.991, Z    +0.000, E1  +350.742, E3 -353323.309}
SPL {X  -159.990, Y  +648.067, Z    +0.000, E1  +342.328, E3 -353327.038}
SPL {X  -159.990, Y  +624.891, Z    +0.000, E1  +327.004, E3 -353345.526}
SPL {X  -159.990, Y  +618.109, Z    +0.000, E1  +324.631, E3 -353353.702}
SPL {X  -159.990, Y  +591.256, Z    +0.000, E1  +319.966, E3 -353397.379}
SPL {X  -159.990, Y  +586.740, Z    +0.000, E1  +319.956, E3 -353408.769}
SPL {X  -159.990, Y  +581.814, Z    +0.000, E1  +319.956, E3 -353421.209}
SPL {X  -159.990, Y  +577.274, Z    +0.000, E1  +319.964, E3 -353432.686}
SPL {X  -159.990, Y  +572.933, Z    +0.000, E1  +319.959, E3 -353443.627}
SPL {X  -159.990, Y  +568.504, Z    +0.000, E1  +319.956, E3 -353454.790}
SPL {X  -159.990, Y  +563.189, Z    +0.000, E1  +319.932, E3 -353468.163}
SPL {X  -159.990, Y  +557.707, Z    +0.000, E1  +319.949, E3 -353482.019}
SPL {X  -159.990, Y  +552.104, Z    +0.000, E1  +319.922, E3 -353496.094}
SPL {X  -159.990, Y  +545.912, Z    +0.000, E1  +319.929, E3 -353511.743}
SPL {X  -159.990, Y  +540.054, Z    +0.000, E1  +319.939, E3 -353526.570}
SPL {X  -159.990, Y  +533.683, Z    +0.000, E1  +319.916, E3 -353542.595}
SPL {X  -159.990, Y  +528.899, Z    +0.000, E1  +319.955, E3 -353554.711}
SPL {X  -159.990, Y  +523.984, Z    +0.000, E1  +319.922, E3 -353567.058}
SPL {X  -159.990, Y  +496.806, Z    +0.000, E1  +312.216, E3 -353580.973}
SPL {X  -159.990, Y  +490.245, Z    +0.000, E1  +312.831, E3 -353597.504}
SPL {X  -159.990, Y  +484.831, Z    +0.000, E1  +314.066, E3 -353615.737}
SPL {X  -159.990, Y  +480.580, Z    +0.000, E1  +315.242, E3 -353631.423}
SPL {X  -159.990, Y  +476.546, Z    +0.000, E1  +316.165, E3 -353645.718}
SPL {X  -159.990, Y  +472.671, Z    +0.000, E1  +317.192, E3 -353660.545}
SPL {X  -159.990, Y  +468.809, Z    +0.000, E1  +318.343, E3 -353676.474}
SPL {X  -159.990, Y  +465.057, Z    +0.000, E1  +319.375, E3 -353691.632}
SPL {X  -159.990, Y  +461.409, Z    +0.000, E1  +319.848, E3 -353703.532}
SPL {X  -159.990, Y  +456.934, Z    +0.000, E1  +319.854, E3 -353714.807}
SPL {X  -159.990, Y  +452.940, Z    +0.000, E1  +319.854, E3 -353724.852}
SPL {X  -159.990, Y  +448.856, Z    +0.000, E1  +319.859, E3 -353735.135}
SPL {X  -159.990, Y  +443.741, Z    +0.000, E1  +319.827, E3 -353747.953}
SPL {X  -159.990, Y  +436.703, Z    +0.000, E1  +319.809, E3 -353765.635}
SPL {X  -159.990, Y  +430.690, Z    +0.000, E1  +319.854, E3 -353780.828}
SPL {X  -159.990, Y  +426.145, Z    +0.000, E1  +319.853, E3 -353792.268}
SPL {X  -159.990, Y  +421.880, Z    +0.000, E1  +319.860, E3 -353803.001}
SPL {X  -159.990, Y  +417.572, Z    +0.000, E1  +319.852, E3 -353813.827}
SPL {X  -159.990, Y  +412.619, Z    +0.000, E1  +319.850, E3 -353826.319}
SPL {X  -159.990, Y  +406.264, Z    +0.000, E1  +319.825, E3 -353842.267}
SPL {X  -159.990, Y  +400.535, Z    +0.000, E1  +319.859, E3 -353856.730}
SPL {X  -159.990, Y  +396.024, Z    +0.000, E1  +319.860, E3 -353868.086}
SPL {X  -159.990, Y  +391.614, Z    +0.000, E1  +319.860, E3 -353879.180}
SPL {X  -159.990, Y  +387.212, Z    +0.000, E1  +319.859, E3 -353890.252}
SPL {X  -159.990, Y  +382.743, Z    +0.000, E1  +319.857, E3 -353901.493}
SPL {X  -159.925, Y  +377.946, Z    +0.000, E1  +319.864, E3 -353913.630}
SPL {X  -159.703, Y  +372.915, Z    +0.000, E1  +319.904, E3 -353926.530}
SPL {X  -159.358, Y  +368.290, Z    +0.000, E1  +319.961, E3 -353938.493}
SPL {X  -158.955, Y  +364.333, Z    +0.000, E1  +320.046, E3 -353948.895}
SPL {X  -158.270, Y  +359.106, Z    +0.000, E1  +320.118, E3 -353962.706}
SPL {X  -157.143, Y  +352.453, Z    +0.000, E1  +320.322, E3 -353980.637}
SPL {X  -156.148, Y  +347.650, Z    +0.000, E1  +320.549, E3 -353993.823}
SPL {X  -155.268, Y  +343.918, Z    +0.000, E1  +320.696, E3 -354004.104}
SPL {X  -154.153, Y  +339.677, Z    +0.000, E1  +320.896, E3 -354015.911}
SPL {X  -152.885, Y  +335.352, Z    +0.000, E1  +321.114, E3 -354028.065}
SPL {X  -151.010, Y  +329.654, Z    +0.000, E1  +326.674, E3 -354088.281}
ENDSPLINE

SPLINE
SPL {X  -157.513, Y  +354.453, Z    +0.000, E1  +340.941, E3 -354134.315}
SPL {X  -159.638, Y  +371.886, Z    +0.000, E1  +350.545, E3 -354144.978}
SPL {X  -159.990, Y  +382.357, Z    +0.000, E1  +356.972, E3 -354148.393}
SPL {X  -159.990, Y  +388.001, Z    +0.000, E1  +361.086, E3 -354149.731}
SPL {X  -159.990, Y  +392.647, Z    +0.000, E1  +364.974, E3 -354150.869}
SPL {X  -159.990, Y  +397.943, Z    +0.000, E1  +369.963, E3 -354152.454}
SPL {X  -159.990, Y  +406.530, Z    +0.000, E1  +377.917, E3 -354156.352}
SPL {X  -159.990, Y  +429.014, Z    +0.000, E1  +392.438, E3 -354175.008}
SPL {X  -159.990, Y  +437.635, Z    +0.000, E1  +395.495, E3 -354185.240}
SPL {X  -159.990, Y  +460.330, Z    +0.000, E1  +398.908, E3 -354225.928}
SPL {X  -159.990, Y  +464.953, Z    +0.000, E1  +398.907, E3 -354238.086}
SPL {X  -159.990, Y  +469.353, Z    +0.000, E1  +398.902, E3 -354249.666}
SPL {X  -159.990, Y  +473.222, Z    +0.000, E1  +398.891, E3 -354259.875}
SPL {X  -159.990, Y  +476.615, Z    +0.000, E1  +398.890, E3 -354268.810}
SPL {X  -159.990, Y  +481.308, Z    +0.000, E1  +398.917, E3 -354281.092}
SPL {X  -159.990, Y  +486.996, Z    +0.000, E1  +398.928, E3 -354296.000}
SPL {X  -159.990, Y  +492.629, Z    +0.000, E1  +398.922, E3 -354310.807}
SPL {X  -159.990, Y  +497.431, Z    +0.000, E1  +398.905, E3 -354323.473}
SPL {X  -159.990, Y  +502.093, Z    +0.000, E1  +398.909, E3 -354335.747}
SPL {X  -159.990, Y  +507.821, Z    +0.000, E1  +398.930, E3 -354350.768}
SPL {X  -159.990, Y  +513.533, Z    +0.000, E1  +398.910, E3 -354365.827}
SPL {X  -159.990, Y  +518.435, Z    +0.000, E1  +398.905, E3 -354378.722}
SPL {X  -159.990, Y  +523.478, Z    +0.000, E1  +398.918, E3 -354391.951}
SPL {X  -159.990, Y  +528.627, Z    +0.000, E1  +398.910, E3 -354405.504}
SPL {X  -159.990, Y  +533.053, Z    +0.000, E1  +398.899, E3 -354417.162}
SPL {X  -159.990, Y  +537.174, Z    +0.000, E1  +398.910, E3 -354427.976}
SPL {X  -159.990, Y  +541.259, Z    +0.000, E1  +398.888, E3 -354438.776}
SPL {X  -159.990, Y  +545.676, Z    +0.000, E1  +398.913, E3 -354450.347}
SPL {X  -159.990, Y  +550.777, Z    +0.000, E1  +398.906, E3 -354463.766}
SPL {X  -159.990, Y  +556.271, Z    +0.000, E1  +398.927, E3 -354478.168}
SPL {X  -159.990, Y  +561.696, Z    +0.000, E1  +398.912, E3 -354492.438}
SPL {X  -159.990, Y  +566.650, Z    +0.000, E1  +398.917, E3 -354505.452}
SPL {X  -159.990, Y  +571.814, Z    +0.000, E1  +398.914, E3 -354519.054}
SPL {X  -159.990, Y  +577.636, Z    +0.000, E1  +398.929, E3 -354534.352}
SPL {X  -159.990, Y  +583.167, Z    +0.000, E1  +398.906, E3 -354548.927}
SPL {X  -159.990, Y  +587.761, Z    +0.000, E1  +398.902, E3 -354561.012}
SPL {X  -159.990, Y  +592.962, Z    +0.000, E1  +398.925, E3 -354574.656}
SPL {X  -159.990, Y  +597.767, Z    +0.000, E1  +398.897, E3 -354587.331}
SPL {X  -159.990, Y  +602.727, Z    +0.000, E1  +398.920, E3 -354600.342}
SPL {X  -159.990, Y  +608.112, Z    +0.000, E1  +398.911, E3 -354614.517}
SPL {X  -159.990, Y  +613.039, Z    +0.000, E1  +398.906, E3 -354627.479}
SPL {X  -159.990, Y  +618.087, Z    +0.000, E1  +398.915, E3 -354640.738}
SPL {X  -159.990, Y  +623.264, Z    +0.000, E1  +398.906, E3 -354654.372}
SPL {X  -159.990, Y  +628.669, Z    +0.000, E1  +398.928, E3 -354668.541}
SPL {X  -159.990, Y  +634.089, Z    +0.000, E1  +398.907, E3 -354682.816}
SPL {X  -159.990, Y  +638.639, Z    +0.000, E1  +398.904, E3 -354694.802}
SPL {X  -159.990, Y  +643.555, Z    +0.000, E1  +398.910, E3 -354707.722}
SPL {X  -159.990, Y  +649.380, Z    +0.000, E1  +398.930, E3 -354723.000}
SPL {X  -159.990, Y  +654.813, Z    +0.000, E1  +398.905, E3 -354737.324}
SPL {X  -159.990, Y  +660.353, Z    +0.000, E1  +398.930, E3 -354751.855}
SPL {X  -159.990, Y  +665.703, Z    +0.000, E1  +398.903, E3 -354765.963}
SPL {X  -159.990, Y  +669.966, Z    +0.000, E1  +398.902, E3 -354777.169}
SPL {X  -159.954, Y  +674.895, Z    +0.000, E1  +398.910, E3 -354790.149}
SPL {X  -159.761, Y  +680.061, Z    +0.000, E1  +398.873, E3 -354803.928}
SPL {X  -159.443, Y  +684.716, Z    +0.000, E1  +398.815, E3 -354816.493}
SPL {X  -158.962, Y  +689.604, Z    +0.000, E1  +398.740, E3 -354829.863}
SPL {X  -158.318, Y  +694.567, Z    +0.000, E1  +398.614, E3 -354843.624}
SPL {X  -157.472, Y  +699.775, Z    +0.000, E1  +398.483, E3 -354858.183}
SPL {X  -156.506, Y  +704.705, Z    +0.000, E1  +398.294, E3 -354872.184}
SPL {X  -155.357, Y  +709.721, Z    +0.000, E1  +398.108, E3 -354886.539}
SPL {X  -154.286, Y  +713.838, Z    +0.000, E1  +397.877, E3 -354898.521}
SPL {X  -153.345, Y  +717.131, Z    +0.000, E1  +397.713, E3 -354908.136}
SPL {X  -151.080, Y  +724.146, Z    +0.000, E1  +393.201, E3 -354966.589}
ENDSPLINE

SPLINE
SPL {X  -157.921, Y  +697.149, Z    +0.000, E1  +377.701, E3 -355018.150}
SPL {X  -159.579, Y  +682.959, Z    +0.000, E1  +369.793, E3 -355026.098}
SPL {X  -159.938, Y  +675.561, Z    +0.000, E1  +365.399, E3 -355028.521}
SPL {X  -159.990, Y  +669.910, Z    +0.000, E1  +361.710, E3 -355029.812}
SPL {X  -159.990, Y  +665.465, Z    +0.000, E1  +358.378, E3 -355030.729}
SPL {X  -159.990, Y  +661.791, Z    +0.000, E1  +355.213, E3 -355031.567}
SPL {X  -159.990, Y  +656.991, Z    +0.000, E1  +350.742, E3 -355032.986}
SPL {X  -159.990, Y  +649.722, Z    +0.000, E1  +343.777, E3 -355035.905}
SPL {X  -159.990, Y  +645.752, Z    +0.000, E1  +340.157, E3 -355037.846}
SPL {X  -159.990, Y  +624.891, Z    +0.000, E1  +327.004, E3 -355055.203}
SPL {X  -159.990, Y  +618.109, Z    +0.000, E1  +324.631, E3 -355063.379}
SPL {X  -159.990, Y  +591.256, Z    +0.000, E1  +319.966, E3 -355107.056}
SPL {X  -159.990, Y  +586.740, Z    +0.000, E1  +319.956, E3 -355118.446}
SPL {X  -159.990, Y  +581.814, Z    +0.000, E1  +319.956, E3 -355130.886}
SPL {X  -159.990, Y  +577.274, Z    +0.000, E1  +319.964, E3 -355142.363}
SPL {X  -159.990, Y  +572.933, Z    +0.000, E1  +319.959, E3 -355153.305}
SPL {X  -159.990, Y  +568.504, Z    +0.000, E1  +319.956, E3 -355164.467}
SPL {X  -159.990, Y  +564.427, Z    +0.000, E1  +319.959, E3 -355174.753}
SPL {X  -159.990, Y  +558.823, Z    +0.000, E1  +319.916, E3 -355188.833}
SPL {X  -159.990, Y  +553.571, Z    +0.000, E1  +319.954, E3 -355202.114}
SPL {X  -159.990, Y  +549.413, Z    +0.000, E1  +319.938, E3 -355212.581}
SPL {X  -159.990, Y  +544.924, Z    +0.000, E1  +319.955, E3 -355223.962}
SPL {X  -159.990, Y  +540.054, Z    +0.000, E1  +319.939, E3 -355236.248}
SPL {X  -159.990, Y  +535.835, Z    +0.000, E1  +319.966, E3 -355246.928}
SPL {X  -159.990, Y  +532.291, Z    +0.000, E1  +319.951, E3 -355255.836}
SPL {X  -159.990, Y  +527.393, Z    +0.000, E1  +319.924, E3 -355268.145}
SPL {X  -159.990, Y  +522.533, Z    +0.000, E1  +319.951, E3 -355280.442}
SPL {X  -159.990, Y  +502.378, Z    +0.000, E1  +313.079, E3 -355284.847}
SPL {X  -159.990, Y  +493.568, Z    +0.000, E1  +312.053, E3 -355296.014}
SPL {X  -159.990, Y  +489.464, Z    +0.000, E1  +313.059, E3 -355309.881}
SPL {X  -159.990, Y  +484.831, Z    +0.000, E1  +314.066, E3 -355325.414}
SPL {X  -159.990, Y  +480.580, Z    +0.000, E1  +315.242, E3 -355341.100}
SPL {X  -159.990, Y  +476.546, Z    +0.000, E1  +316.165, E3 -355355.395}
SPL {X  -159.990, Y  +473.377, Z    +0.000, E1  +316.953, E3 -355367.010}
SPL {X  -159.990, Y  +470.788, Z    +0.000, E1  +317.853, E3 -355378.423}
SPL {X  -159.990, Y  +467.944, Z    +0.000, E1  +318.635, E3 -355389.744}
SPL {X  -159.990, Y  +465.057, Z    +0.000, E1  +319.375, E3 -355401.309}
SPL {X  -159.990, Y  +461.409, Z    +0.000, E1  +319.848, E3 -355413.209}
SPL {X  -159.990, Y  +456.934, Z    +0.000, E1  +319.854, E3 -355424.485}
SPL {X  -159.990, Y  +452.940, Z    +0.000, E1  +319.854, E3 -355434.529}
SPL {X  -159.990, Y  +448.856, Z    +0.000, E1  +319.859, E3 -355444.813}
SPL {X  -159.990, Y  +443.741, Z    +0.000, E1  +319.827, E3 -355457.630}
SPL {X  -159.990, Y  +436.703, Z    +0.000, E1  +319.809, E3 -355475.312}
SPL {X  -159.990, Y  +430.690, Z    +0.000, E1  +319.854, E3 -355490.505}
SPL {X  -159.990, Y  +426.145, Z    +0.000, E1  +319.853, E3 -355501.945}
SPL {X  -159.990, Y  +421.880, Z    +0.000, E1  +319.860, E3 -355512.678}
SPL {X  -159.990, Y  +417.572, Z    +0.000, E1  +319.852, E3 -355523.505}
SPL {X  -159.990, Y  +412.619, Z    +0.000, E1  +319.850, E3 -355535.996}
SPL {X  -159.990, Y  +408.586, Z    +0.000, E1  +319.876, E3 -355546.181}
SPL {X  -159.990, Y  +404.988, Z    +0.000, E1  +319.861, E3 -355555.209}
SPL {X  -159.990, Y  +400.535, Z    +0.000, E1  +319.859, E3 -355566.407}
SPL {X  -159.990, Y  +396.024, Z    +0.000, E1  +319.860, E3 -355577.763}
SPL {X  -159.990, Y  +391.614, Z    +0.000, E1  +319.860, E3 -355588.857}
SPL {X  -159.990, Y  +387.212, Z    +0.000, E1  +319.859, E3 -355599.929}
SPL {X  -159.990, Y  +382.743, Z    +0.000, E1  +319.857, E3 -355611.171}
SPL {X  -159.925, Y  +377.946, Z    +0.000, E1  +319.864, E3 -355623.308}
SPL {X  -159.703, Y  +372.915, Z    +0.000, E1  +319.904, E3 -355636.207}
SPL {X  -159.358, Y  +368.290, Z    +0.000, E1  +319.961, E3 -355648.170}
SPL {X  -158.955, Y  +364.333, Z    +0.000, E1  +320.046, E3 -355658.572}
SPL {X  -158.482, Y  +360.589, Z    +0.000, E1  +320.125, E3 -355668.499}
SPL {X  -157.729, Y  +355.695, Z    +0.000, E1  +320.237, E3 -355681.571}
SPL {X  -156.893, Y  +351.173, Z    +0.000, E1  +320.410, E3 -355693.855}
SPL {X  -156.148, Y  +347.650, Z    +0.000, E1  +320.549, E3 -355703.501}
SPL {X  -155.268, Y  +343.918, Z    +0.000, E1  +320.696, E3 -355713.781}
SPL {X  -153.936, Y  +338.906, Z    +0.000, E1  +320.911, E3 -355727.721}
SPL {X  -152.628, Y  +334.526, Z    +0.000, E1  +321.188, E3 -355740.123}
SPL {X  -151.010, Y  +329.654, Z    +0.000, E1  +326.674, E3 -355797.959}
ENDSPLINE

SPLINE
SPL {X  -157.513, Y  +354.453, Z    +0.000, E1  +340.941, E3 -355843.993}
SPL {X  -159.408, Y  +368.861, Z    +0.000, E1  +348.865, E3 -355853.416}
SPL {X  -159.941, Y  +378.532, Z    +0.000, E1  +354.551, E3 -355857.021}
SPL {X  -159.990, Y  +383.966, Z    +0.000, E1  +358.149, E3 -355858.473}
SPL {X  -159.990, Y  +388.001, Z    +0.000, E1  +361.086, E3 -355859.408}
SPL {X  -159.990, Y  +392.647, Z    +0.000, E1  +364.974, E3 -355860.547}
SPL {X  -159.990, Y  +397.943, Z    +0.000, E1  +369.963, E3 -355862.131}
SPL {X  -159.990, Y  +406.530, Z    +0.000, E1  +377.917, E3 -355866.029}
SPL {X  -159.990, Y  +429.014, Z    +0.000, E1  +392.438, E3 -355884.686}
SPL {X  -159.990, Y  +437.635, Z    +0.000, E1  +395.495, E3 -355894.918}
SPL {X  -159.990, Y  +460.330, Z    +0.000, E1  +398.908, E3 -355935.605}
SPL {X  -159.990, Y  +464.953, Z    +0.000, E1  +398.907, E3 -355947.764}
SPL {X  -159.990, Y  +469.353, Z    +0.000, E1  +398.902, E3 -355959.344}
SPL {X  -159.990, Y  +475.034, Z    +0.000, E1  +398.936, E3 -355974.259}
SPL {X  -159.990, Y  +481.308, Z    +0.000, E1  +398.917, E3 -355990.770}
SPL {X  -159.990, Y  +486.996, Z    +0.000, E1  +398.928, E3 -356005.677}
SPL {X  -159.990, Y  +492.629, Z    +0.000, E1  +398.922, E3 -356020.484}
SPL {X  -159.990, Y  +497.431, Z    +0.000, E1  +398.905, E3 -356033.150}
SPL {X  -159.990, Y  +502.093, Z    +0.000, E1  +398.909, E3 -356045.425}
SPL {X  -159.990, Y  +507.821, Z    +0.000, E1  +398.930, E3 -356060.445}
SPL {X  -159.990, Y  +513.533, Z    +0.000, E1  +398.910, E3 -356075.504}
SPL {X  -159.990, Y  +518.435, Z    +0.000, E1  +398.905, E3 -356088.400}
SPL {X  -159.990, Y  +523.478, Z    +0.000, E1  +398.918, E3 -356101.628}
SPL {X  -159.990, Y  +528.627, Z    +0.000, E1  +398.910, E3 -356115.182}
SPL {X  -159.990, Y  +534.392, Z    +0.000, E1  +398.932, E3 -356130.312}
SPL {X  -159.990, Y  +540.299, Z    +0.000, E1  +398.912, E3 -356145.886}
SPL {X  -159.990, Y  +545.676, Z    +0.000, E1  +398.913, E3 -356160.024}
SPL {X  -159.990, Y  +550.777, Z    +0.000, E1  +398.906, E3 -356173.443}
SPL {X  -159.990, Y  +556.271, Z    +0.000, E1  +398.927, E3 -356187.846}
SPL {X  -159.990, Y  +561.696, Z    +0.000, E1  +398.912, E3 -356202.115}
SPL {X  -159.990, Y  +566.650, Z    +0.000, E1  +398.917, E3 -356215.129}
SPL {X  -159.990, Y  +571.814, Z    +0.000, E1  +398.914, E3 -356228.732}
SPL {X  -159.990, Y  +577.636, Z    +0.000, E1  +398.929, E3 -356244.029}
SPL {X  -159.990, Y  +583.167, Z    +0.000, E1  +398.906, E3 -356258.605}
SPL {X  -159.990, Y  +589.106, Z    +0.000, E1  +398.939, E3 -356274.172}
SPL {X  -159.990, Y  +596.185, Z    +0.000, E1  +398.945, E3 -356292.780}
SPL {X  -159.990, Y  +602.727, Z    +0.000, E1  +398.920, E3 -356310.020}
SPL {X  -159.990, Y  +608.112, Z    +0.000, E1  +398.911, E3 -356324.194}
SPL {X  -159.990, Y  +614.125, Z    +0.000, E1  +398.936, E3 -356339.969}
SPL {X  -159.990, Y  +619.061, Z    +0.000, E1  +398.894, E3 -356353.001}
SPL {X  -159.990, Y  +623.264, Z    +0.000, E1  +398.906, E3 -356364.050}
SPL {X  -159.990, Y  +628.669, Z    +0.000, E1  +398.928, E3 -356378.218}
SPL {X  -159.990, Y  +634.089, Z    +0.000, E1  +398.907, E3 -356392.494}
SPL {X  -159.990, Y  +638.639, Z    +0.000, E1  +398.904, E3 -356404.479}
SPL {X  -159.990, Y  +644.750, Z    +0.000, E1  +398.946, E3 -356420.485}
SPL {X  -159.990, Y  +650.458, Z    +0.000, E1  +398.900, E3 -356435.557}
SPL {X  -159.990, Y  +654.813, Z    +0.000, E1  +398.905, E3 -356447.001}
SPL {X  -159.990, Y  +660.353, Z    +0.000, E1  +398.930, E3 -356461.533}
SPL {X  -159.990, Y  +665.703, Z    +0.000, E1  +398.903, E3 -356475.640}
SPL {X  -159.990, Y  +671.472, Z    +0.000, E1  +398.942, E3 -356490.745}
SPL {X  -159.920, Y  +676.216, Z    +0.000, E1  +398.875, E3 -356503.380}
SPL {X  -159.761, Y  +680.061, Z    +0.000, E1  +398.873, E3 -356513.606}
SPL {X  -159.443, Y  +684.716, Z    +0.000, E1  +398.815, E3 -356526.171}
SPL {X  -158.962, Y  +689.604, Z    +0.000, E1  +398.740, E3 -356539.540}
SPL {X  -158.139, Y  +695.766, Z    +0.000, E1  +398.623, E3 -356556.586}
SPL {X  -157.275, Y  +700.848, Z    +0.000, E1  +398.415, E3 -356570.938}
SPL {X  -156.506, Y  +704.705, Z    +0.000, E1  +398.294, E3 -356581.861}
SPL {X  -155.357, Y  +709.721, Z    +0.000, E1  +398.108, E3 -356596.216}
SPL {X  -154.286, Y  +713.838, Z    +0.000, E1  +397.877, E3 -356608.199}
SPL {X  -153.345, Y  +717.131, Z    +0.000, E1  +397.713, E3 -356617.813}
SPL {X  -151.080, Y  +724.146, Z    +0.000, E1  +393.201, E3 -356676.267}
ENDSPLINE

SPLINE
SPL {X  -157.921, Y  +697.149, Z    +0.000, E1  +377.701, E3 -356727.828}
SPL {X  -159.579, Y  +682.959, Z    +0.000, E1  +369.793, E3 -356735.776}
SPL {X  -159.938, Y  +675.561, Z    +0.000, E1  +365.399, E3 -356738.198}
SPL {X  -159.990, Y  +669.910, Z    +0.000, E1  +361.710, E3 -356739.489}
SPL {X  -159.990, Y  +665.465, Z    +0.000, E1  +358.378, E3 -356740.406}
SPL {X  -159.990, Y  +661.791, Z    +0.000, E1  +355.213, E3 -356741.244}
SPL {X  -159.990, Y  +656.991, Z    +0.000, E1  +350.742, E3 -356742.663}
SPL {X  -159.990, Y  +648.067, Z    +0.000, E1  +342.328, E3 -356746.393}
SPL {X  -159.990, Y  +624.891, Z    +0.000, E1  +327.004, E3 -356764.881}
SPL {X  -159.990, Y  +618.109, Z    +0.000, E1  +324.631, E3 -356773.057}
SPL {X  -159.990, Y  +591.256, Z    +0.000, E1  +319.966, E3 -356816.734}
SPL {X  -159.990, Y  +586.740, Z    +0.000, E1  +319.956, E3 -356828.124}
SPL {X  -159.990, Y  +581.814, Z    +0.000, E1  +319.956, E3 -356840.563}
SPL {X  -159.990, Y  +577.274, Z    +0.000, E1  +319.964, E3 -356852.041}
SPL {X  -159.990, Y  +572.933, Z    +0.000, E1  +319.959, E3 -356862.982}
SPL {X  -159.990, Y  +568.504, Z    +0.000, E1  +319.956, E3 -356874.145}
SPL {X  -159.990, Y  +563.189, Z    +0.000, E1  +319.932, E3 -356887.518}
SPL {X  -159.990, Y  +557.707, Z    +0.000, E1  +319.949, E3 -356901.373}
SPL {X  -159.990, Y  +552.104, Z    +0.000, E1  +319.922, E3 -356915.448}
SPL {X  -159.990, Y  +545.912, Z    +0.000, E1  +319.929, E3 -356931.098}
SPL {X  -159.990, Y  +540.054, Z    +0.000, E1  +319.939, E3 -356945.925}
SPL {X  -159.990, Y  +533.683, Z    +0.000, E1  +319.916, E3 -356961.950}
SPL {X  -159.990, Y  +528.899, Z    +0.000, E1  +319.955, E3 -356974.066}
SPL {X  -159.990, Y  +523.984, Z    +0.000, E1  +319.922, E3 -356986.413}
SPL {X  -159.990, Y  +496.806, Z    +0.000, E1  +312.216, E3 -357000.327}
SPL {X  -159.990, Y  +490.245, Z    +0.000, E1  +312.831, E3 -357016.859}
SPL {X  -159.990, Y  +484.831, Z    +0.000, E1  +314.066, E3 -357035.091}
SPL {X  -159.990, Y  +480.580, Z    +0.000, E1  +315.242, E3 -357050.778}
SPL {X  -159.990, Y  +476.546, Z    +0.000, E1  +316.165, E3 -357065.073}
SPL {X  -159.990, Y  +472.671, Z    +0.000, E1  +317.192, E3 -357079.900}
SPL {X  -159.990, Y  +468.809, Z    +0.000, E1  +318.343, E3 -357095.828}
SPL {X  -159.990, Y  +465.057, Z    +0.000, E1  +319.375, E3 -357110.987}
SPL {X  -159.990, Y  +461.409, Z    +0.000, E1  +319.848, E3 -357122.886}
SPL {X  -159.990, Y  +456.934, Z    +0.000, E1  +319.854, E3 -357134.162}
SPL {X  -159.990, Y  +452.940, Z    +0.000, E1  +319.854, E3 -357144.207}
SPL {X  -159.990, Y  +448.856, Z    +0.000, E1  +319.859, E3 -357154.490}
SPL {X  -159.990, Y  +443.741, Z    +0.000, E1  +319.827, E3 -357167.308}
SPL {X  -159.990, Y  +436.703, Z    +0.000, E1  +319.809, E3 -357184.990}
SPL {X  -159.990, Y  +430.690, Z    +0.000, E1  +319.854, E3 -357200.183}
SPL {X  -159.990, Y  +426.145, Z    +0.000, E1  +319.853, E3 -357211.623}
SPL {X  -159.990, Y  +421.880, Z    +0.000, E1  +319.860, E3 -357222.356}
SPL {X  -159.990, Y  +417.572, Z    +0.000, E1  +319.852, E3 -357233.182}
SPL {X  -159.990, Y  +412.619, Z    +0.000, E1  +319.850, E3 -357245.674}
SPL {X  -159.990, Y  +406.264, Z    +0.000, E1  +319.825, E3 -357261.622}
SPL {X  -159.990, Y  +400.535, Z    +0.000, E1  +319.859, E3 -357276.085}
SPL {X  -159.990, Y  +396.024, Z    +0.000, E1  +319.860, E3 -357287.441}
SPL {X  -159.990, Y  +391.614, Z    +0.000, E1  +319.860, E3 -357298.534}
SPL {X  -159.990, Y  +387.212, Z    +0.000, E1  +319.859, E3 -357309.607}
SPL {X  -159.990, Y  +382.743, Z    +0.000, E1  +319.857, E3 -357320.848}
SPL {X  -159.925, Y  +377.946, Z    +0.000, E1  +319.864, E3 -357332.985}
SPL {X  -159.703, Y  +372.915, Z    +0.000, E1  +319.904, E3 -357345.885}
SPL {X  -159.358, Y  +368.290, Z    +0.000, E1  +319.961, E3 -357357.847}
SPL {X  -158.955, Y  +364.333, Z    +0.000, E1  +320.046, E3 -357368.250}
SPL {X  -158.270, Y  +359.106, Z    +0.000, E1  +320.118, E3 -357382.061}
SPL {X  -157.143, Y  +352.453, Z    +0.000, E1  +320.322, E3 -357399.992}
SPL {X  -156.148, Y  +347.650, Z    +0.000, E1  +320.549, E3 -357413.178}
SPL {X  -155.268, Y  +343.918, Z    +0.000, E1  +320.696, E3 -357423.459}
SPL {X  -154.153, Y  +339.677, Z    +0.000, E1  +320.896, E3 -357435.266}
SPL {X  -152.885, Y  +335.352, Z    +0.000, E1  +321.114, E3 -357447.420}
SPL {X  -151.010, Y  +329.654, Z    +0.000, E1  +326.674, E3 -357507.636}
ENDSPLINE

SPLINE
SPL {X  -157.513, Y  +354.453, Z    +0.000, E1  +340.941, E3 -357553.670}
SPL {X  -159.638, Y  +371.886, Z    +0.000, E1  +350.545, E3 -357564.332}
SPL {X  -159.990, Y  +382.357, Z    +0.000, E1  +356.972, E3 -357567.748}
SPL {X  -159.990, Y  +388.001, Z    +0.000, E1  +361.086, E3 -357569.086}
SPL {X  -159.990, Y  +392.647, Z    +0.000, E1  +364.974, E3 -357570.224}
SPL {X  -159.990, Y  +397.943, Z    +0.000, E1  +369.963, E3 -357571.809}
SPL {X  -159.990, Y  +406.530, Z    +0.000, E1  +377.917, E3 -357575.707}
SPL {X  -159.990, Y  +429.014, Z    +0.000, E1  +392.438, E3 -357594.363}
SPL {X  -159.990, Y  +437.635, Z    +0.000, E1  +395.495, E3 -357604.595}
SPL {X  -159.990, Y  +460.330, Z    +0.000, E1  +398.908, E3 -357645.283}
SPL {X  -159.990, Y  +464.953, Z    +0.000, E1  +398.907, E3 -357657.441}
SPL {X  -159.990, Y  +469.353, Z    +0.000, E1  +398.902, E3 -357669.021}
SPL {X  -159.990, Y  +473.222, Z    +0.000, E1  +398.891, E3 -357679.230}
SPL {X  -159.990, Y  +476.615, Z    +0.000, E1  +398.890, E3 -357688.165}
SPL {X  -159.990, Y  +481.308, Z    +0.000, E1  +398.917, E3 -357700.447}
SPL {X  -159.990, Y  +486.996, Z    +0.000, E1  +398.928, E3 -357715.355}
SPL {X  -159.990, Y  +492.629, Z    +0.000, E1  +398.922, E3 -357730.162}
SPL {X  -159.990, Y  +497.431, Z    +0.000, E1  +398.905, E3 -357742.828}
SPL {X  -159.990, Y  +502.093, Z    +0.000, E1  +398.909, E3 -357755.102}
SPL {X  -159.990, Y  +507.821, Z    +0.000, E1  +398.930, E3 -357770.122}
SPL {X  -159.990, Y  +513.533, Z    +0.000, E1  +398.910, E3 -357785.182}
SPL {X  -159.990, Y  +518.435, Z    +0.000, E1  +398.905, E3 -357798.077}
SPL {X  -159.990, Y  +523.478, Z    +0.000, E1  +398.918, E3 -357811.305}
SPL {X  -159.990, Y  +528.627, Z    +0.000, E1  +398.910, E3 -357824.859}
SPL {X  -159.990, Y  +534.392, Z    +0.000, E1  +398.932, E3 -357839.989}
SPL {X  -159.990, Y  +540.299, Z    +0.000, E1  +398.912, E3 -357855.564}
SPL {X  -159.990, Y  +545.676, Z    +0.000, E1  +398.913, E3 -357869.702}
SPL {X  -159.990, Y  +550.777, Z    +0.000, E1  +398.906, E3 -357883.121}
SPL {X  -159.990, Y  +556.271, Z    +0.000, E1  +398.927, E3 -357897.523}
SPL {X  -159.990, Y  +561.696, Z    +0.000, E1  +398.912, E3 -357911.793}
SPL {X  -159.990, Y  +566.650, Z    +0.000, E1  +398.917, E3 -357924.806}
SPL {X  -159.990, Y  +571.814, Z    +0.000, E1  +398.914, E3 -357938.409}
SPL {X  -159.990, Y  +576.364, Z    +0.000, E1  +398.896, E3 -357950.412}
SPL {X  -159.990, Y  +582.060, Z    +0.000, E1  +398.942, E3 -357965.318}
SPL {X  -159.990, Y  +587.761, Z    +0.000, E1  +398.902, E3 -357980.367}
SPL {X  -159.990, Y  +592.962, Z    +0.000, E1  +398.925, E3 -357994.011}
SPL {X  -159.990, Y  +597.767, Z    +0.000, E1  +398.897, E3 -358006.686}
SPL {X  -159.990, Y  +602.727, Z    +0.000, E1  +398.920, E3 -358019.697}
SPL {X  -159.990, Y  +608.112, Z    +0.000, E1  +398.911, E3 -358033.872}
SPL {X  -159.990, Y  +614.125, Z    +0.000, E1  +398.936, E3 -358049.647}
SPL {X  -159.990, Y  +619.061, Z    +0.000, E1  +398.894, E3 -358062.678}
SPL {X  -159.990, Y  +623.264, Z    +0.000, E1  +398.906, E3 -358073.727}
SPL {X  -159.990, Y  +627.067, Z    +0.000, E1  +398.891, E3 -358083.747}
SPL {X  -159.990, Y  +630.187, Z    +0.000, E1  +398.892, E3 -358091.935}
SPL {X  -159.990, Y  +634.089, Z    +0.000, E1  +398.907, E3 -358102.171}
SPL {X  -159.990, Y  +638.639, Z    +0.000, E1  +398.904, E3 -358114.157}
SPL {X  -159.990, Y  +643.555, Z    +0.000, E1  +398.910, E3 -358127.077}
SPL {X  -159.990, Y  +649.380, Z    +0.000, E1  +398.930, E3 -358142.354}
SPL {X  -159.990, Y  +654.813, Z    +0.000, E1  +398.905, E3 -358156.679}
SPL {X  -159.990, Y  +658.715, Z    +0.000, E1  +398.892, E3 -358166.960}
SPL {X  -159.990, Y  +661.848, Z    +0.000, E1  +398.892, E3 -358175.198}
SPL {X  -159.990, Y  +665.703, Z    +0.000, E1  +398.903, E3 -358185.318}
SPL {X  -159.990, Y  +669.966, Z    +0.000, E1  +398.902, E3 -358196.524}
SPL {X  -159.954, Y  +674.895, Z    +0.000, E1  +398.910, E3 -358209.504}
SPL {X  -159.761, Y  +680.061, Z    +0.000, E1  +398.873, E3 -358223.283}
SPL {X  -159.443, Y  +684.716, Z    +0.000, E1  +398.815, E3 -358235.848}
SPL {X  -158.962, Y  +689.604, Z    +0.000, E1  +398.740, E3 -358249.217}
SPL {X  -158.139, Y  +695.766, Z    +0.000, E1  +398.623, E3 -358266.263}
SPL {X  -157.275, Y  +700.848, Z    +0.000, E1  +398.415, E3 -358280.615}
SPL {X  -156.506, Y  +704.705, Z    +0.000, E1  +398.294, E3 -358291.539}
SPL {X  -155.357, Y  +709.721, Z    +0.000, E1  +398.108, E3 -358305.894}
SPL {X  -154.286, Y  +713.838, Z    +0.000, E1  +397.877, E3 -358317.876}
SPL {X  -153.345, Y  +717.131, Z    +0.000, E1  +397.713, E3 -358327.490}
SPL {X  -151.080, Y  +724.146, Z    +0.000, E1  +393.201, E3 -358385.944}
ENDSPLINE

